Yaskawa INFORM job: pointsclTRJ3.JBI

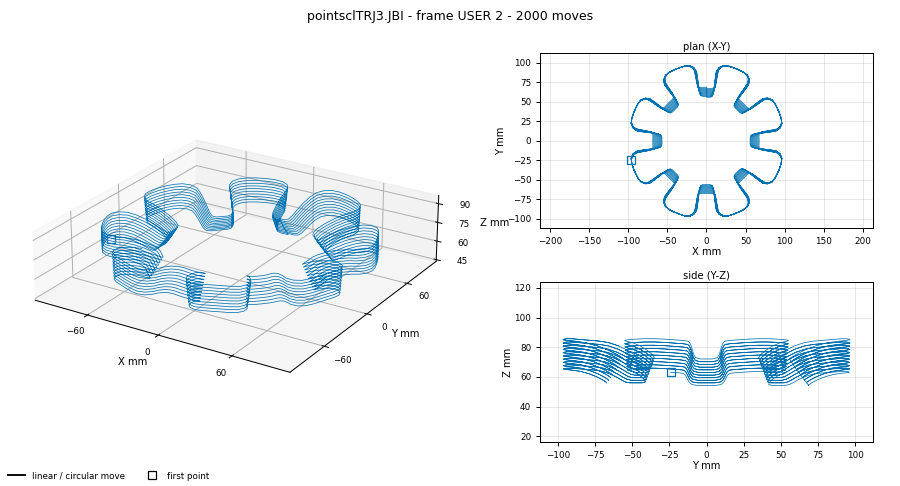
[picture p0: tool path of pointsclTRJ3.JBI in frame USER 2, 2000 of 2000 moves have a stored position in this frame; points joined in program order, loops and branches not executed]
/JOB
//NAME pointsclTRJ3
//POS
///NPOS 2000,0,0,0,0,0
///USER 2
///TOOL 1
///POSTYPE USER
///RECTAN
///RCONF 1,0,0,0,0,0,0,0,0,0,0,0,0,0,0,0,0,0,0,0,0,0,0,0
C00000=-96.154,-24.159,63.210,179.4924,-0.1709,0.0000
C00001=-94.423,-19.246,62.877,-176.7976,1.2873,0.0000
C00002=-90.636,-15.942,62.469,-165.8559,10.6912,0.0000
C00003=-85.405,-14.621,61.698,-164.6923,28.3238,0.0000
C00004=-79.780,-13.569,60.151,-168.6489,33.5433,0.0000
C00005=-74.809,-12.586,58.158,-171.6165,35.6488,0.0000
C00006=-71.127,-11.507,56.252,-173.9501,36.7948,0.0000
C00007=-69.044,-9.699,54.888,-176.7981,37.7947,0.0000
C00008=-68.619,-6.200,54.350,178.5963,38.6094,0.0000
C00009=-68.781,-2.945,54.326,177.6722,38.7088,0.0000
C00010=-68.843,0.000,54.342,179.9995,38.7580,0.0000
C00011=-68.781,2.945,54.326,-177.6718,38.7088,0.0000
C00012=-68.619,6.200,54.350,-178.5977,38.6093,0.0000
C00013=-69.044,9.699,54.888,176.7976,37.7946,0.0000
C00014=-71.127,11.507,56.252,173.9499,36.7948,0.0000
C00015=-74.809,12.586,58.158,171.6165,35.6489,0.0000
C00016=-79.780,13.569,60.151,168.6492,33.5435,0.0000
C00017=-85.405,14.621,61.698,164.6926,28.3243,0.0000
C00018=-90.636,15.942,62.469,165.8558,10.6913,0.0000
C00019=-94.423,19.246,62.877,176.7976,1.2873,0.0000
C00020=-96.154,24.159,63.210,-179.4924,-0.1709,0.0000
C00021=-95.429,29.718,63.547,-178.6193,-0.4469,0.0000
C00022=-93.512,35.416,63.770,-178.6260,-0.4442,0.0000
C00023=-91.166,41.080,63.770,178.7143,0.6573,0.0000
C00024=-88.493,46.465,63.547,178.7076,0.6602,0.0000
C00025=-85.074,50.908,63.210,179.5202,0.2381,0.0000
C00026=-80.376,53.158,62.877,-176.8246,-1.3526,0.0000
C00027=-75.362,52.817,62.469,-162.4707,-2.2128,0.0000
C00028=-70.729,50.052,61.698,-149.5155,9.8553,0.0000
C00029=-66.007,46.818,60.151,-148.1972,15.9457,0.0000
C00030=-61.798,43.998,58.158,-148.3322,19.1679,0.0000
C00031=-58.431,42.158,56.252,-148.7511,21.3364,0.0000
C00032=-55.679,41.963,54.888,-149.5105,23.7114,0.0000
C00033=-52.905,44.137,54.350,-151.2990,27.0505,0.0000
C00034=-50.718,46.553,54.326,-151.7019,27.6849,0.0000
C00035=-48.679,48.679,54.342,-150.4177,26.2748,0.0000
C00036=-46.553,50.718,54.326,-149.2095,24.8209,0.0000
C00037=-44.137,52.905,54.350,-149.7945,25.3228,0.0000
C00038=-41.963,55.680,54.888,-152.9932,27.6813,0.0000
C00039=-42.158,58.431,56.252,-155.4443,28.8948,0.0000
C00040=-43.998,61.798,58.158,-157.7838,29.7283,0.0000
C00041=-46.818,66.007,60.151,-161.4173,30.4455,0.0000
C00042=-50.052,70.729,61.698,-168.6017,29.9881,0.0000
C00043=-52.817,75.362,62.469,177.6796,17.5160,0.0000
C00044=-53.158,80.376,62.877,178.6453,3.1745,0.0000
C00045=-50.908,85.074,63.210,-179.7619,-0.4798,0.0000
C00046=-46.465,88.493,63.547,-179.3396,-1.2923,0.0000
C00047=-41.080,91.166,63.770,-179.3425,-1.2856,0.0000
C00048=-35.416,93.512,63.770,179.5557,1.3739,0.0000
C00049=-29.718,95.429,63.547,179.5530,1.3807,0.0000
C00050=-24.159,96.154,63.210,179.8291,0.5076,0.0000
C00051=-19.246,94.423,62.877,-178.7107,-3.2015,0.0000
C00052=-15.942,90.636,62.469,-168.9825,-13.8937,0.0000
C00053=-14.621,85.405,61.698,-150.8028,-13.4378,0.0000
C00054=-13.569,79.780,60.151,-145.9333,-9.4414,0.0000
C00055=-12.586,74.809,58.158,-144.0591,-6.8041,0.0000
C00056=-11.507,71.127,56.252,-143.0516,-4.8416,0.0000
C00057=-9.699,69.044,54.888,-142.1620,-2.5301,0.0000
C00058=-6.200,68.619,54.350,-141.3823,1.0957,0.0000
C00059=-2.945,68.781,54.326,-141.2681,1.8166,0.0000
C00060=0.000,68.843,54.342,-141.2420,-0.0004,0.0000
C00061=0.000,67.469,56.061,-141.4823,-0.0004,0.0000
C00062=2.820,67.413,56.044,-141.5076,-1.7803,0.0000
C00063=5.989,67.263,56.069,-141.6204,-1.0470,0.0000
C00064=9.441,67.734,56.637,-142.4011,2.5965,0.0000
C00065=11.191,69.937,58.076,-143.2756,4.8842,0.0000
C00066=12.227,73.809,60.085,-144.2799,6.8707,0.0000
C00067=13.183,79.025,62.181,-146.2548,9.6475,0.0000
C00068=14.211,84.918,63.804,-151.9178,13.9840,0.0000
C00069=15.500,90.396,64.610,-174.0678,10.2549,0.0000
C00070=18.832,94.373,65.037,-179.6142,1.0976,0.0000
C00071=23.832,96.213,65.385,179.4380,-1.8355,0.0000
C00072=29.513,95.497,65.736,179.2660,-2.4590,0.0000
C00073=35.347,93.539,65.969,179.2991,-2.3370,0.0000
C00074=41.148,91.136,65.969,-178.8422,2.1478,0.0000
C00075=46.658,88.395,65.736,-178.7792,2.2574,0.0000
C00076=51.181,84.885,65.385,-179.0990,1.6951,0.0000
C00077=53.416,80.048,65.037,179.4966,-1.0488,0.0000
C00078=52.959,74.880,64.610,176.8438,-11.4082,0.0000
C00079=49.997,70.095,63.804,-169.9244,-29.5953,0.0000
C00080=46.557,65.200,62.181,-161.8493,-30.3808,0.0000
C00081=43.545,60.837,60.085,-158.0240,-29.6337,0.0000
C00082=41.540,57.367,58.076,-155.6702,-28.7832,0.0000
C00083=41.220,54.571,56.637,-153.2495,-27.5820,0.0000
C00084=43.327,51.796,56.069,-150.0357,-25.2157,0.0000
C00085=45.674,49.662,56.044,-149.4431,-24.7040,0.0000
C00086=47.708,47.708,56.061,-150.6283,-26.1262,0.0000
C00087=49.662,45.674,56.044,-151.8880,-27.5079,0.0000
C00088=51.797,43.327,56.069,-151.4729,-26.8626,0.0000
C00089=54.571,41.220,56.637,-149.6723,-23.5122,0.0000
C00090=57.367,41.540,58.076,-148.9134,-21.1668,0.0000
C00091=60.837,43.545,60.085,-148.4738,-18.9821,0.0000
C00092=65.200,46.557,62.181,-148.3277,-15.5897,0.0000
C00093=70.095,49.997,63.804,-150.0206,-8.7507,0.0000
C00094=74.880,52.959,64.610,-168.5749,3.0938,0.0000
C00095=80.048,53.416,65.037,-178.9511,0.5034,0.0000
C00096=84.885,51.181,65.385,178.3047,-0.9006,0.0000
C00097=88.395,46.658,65.736,177.7421,-1.2198,0.0000
C00098=91.136,41.148,65.969,177.8518,-1.1570,0.0000
C00099=93.539,35.347,65.969,-177.6628,0.7003,0.0000
C00100=95.497,29.513,65.736,-177.5408,0.7334,0.0000
C00101=96.213,23.832,65.385,-178.1644,0.5617,0.0000
C00102=94.373,18.832,65.037,178.9024,-0.3857,0.0000
C00103=90.396,15.500,64.610,169.6911,-5.8371,0.0000
C00104=84.918,14.211,63.804,164.2377,-27.1799,0.0000
C00105=79.025,13.183,62.181,168.4460,-33.2056,0.0000
C00106=73.809,12.227,60.085,171.5581,-35.4248,0.0000
C00107=69.937,11.191,58.076,173.9145,-36.5694,0.0000
C00108=67.734,9.441,56.637,176.7241,-37.5536,0.0000
C00109=67.263,5.989,56.069,-178.6645,-38.3720,0.0000
C00110=67.413,2.820,56.044,-177.7259,-38.4704,0.0000
C00111=67.469,0.000,56.061,-179.9994,-38.5177,0.0000
C00112=67.413,-2.820,56.044,177.7254,-38.4704,0.0000
C00113=67.263,-5.989,56.069,178.6660,-38.3719,0.0000
C00114=67.734,-9.441,56.637,-176.7236,-37.5535,0.0000
C00115=69.937,-11.191,58.076,-173.9143,-36.5693,0.0000
C00116=73.809,-12.227,60.085,-171.5581,-35.4248,0.0000
C00117=79.025,-13.183,62.181,-168.4462,-33.2058,0.0000
C00118=84.918,-14.211,63.804,-164.2380,-27.1806,0.0000
C00119=90.396,-15.500,64.610,-169.6911,-5.8371,0.0000
C00120=94.373,-18.832,65.037,-178.9024,-0.3857,0.0000
C00121=96.213,-23.832,65.385,178.1644,0.5617,0.0000
C00122=95.497,-29.513,65.736,177.5408,0.7334,0.0000
C00123=93.539,-35.347,65.969,177.6628,0.7003,0.0000
C00124=91.136,-41.148,65.969,-177.8518,-1.1570,0.0000
C00125=88.395,-46.658,65.736,-177.7421,-1.2198,0.0000
C00126=84.885,-51.181,65.385,-178.3047,-0.9006,0.0000
C00127=80.048,-53.416,65.037,178.9511,0.5034,0.0000
C00128=74.880,-52.959,64.610,168.5749,3.0938,0.0000
C00129=70.095,-49.997,63.804,150.0208,-8.7500,0.0000
C00130=65.200,-46.557,62.181,148.3277,-15.5894,0.0000
C00131=60.837,-43.545,60.085,148.4738,-18.9821,0.0000
C00132=57.367,-41.540,58.076,148.9135,-21.1669,0.0000
C00133=54.571,-41.220,56.637,149.6725,-23.5126,0.0000
C00134=51.796,-43.327,56.069,151.4737,-26.8636,0.0000
C00135=49.662,-45.674,56.044,151.8878,-27.5076,0.0000
C00136=47.708,-47.708,56.061,150.6289,-26.1269,0.0000
C00137=45.674,-49.662,56.044,149.4428,-24.7037,0.0000
C00138=43.327,-51.797,56.069,150.0365,-25.2165,0.0000
C00139=41.220,-54.571,56.637,153.2499,-27.5823,0.0000
C00140=41.540,-57.367,58.076,155.6703,-28.7832,0.0000
C00141=43.545,-60.837,60.085,158.0240,-29.6337,0.0000
C00142=46.557,-65.200,62.181,161.8489,-30.3807,0.0000
C00143=49.997,-70.095,63.804,169.9236,-29.5954,0.0000
C00144=52.959,-74.880,64.610,-176.8438,-11.4082,0.0000
C00145=53.416,-80.048,65.037,-179.4966,-1.0488,0.0000
C00146=51.181,-84.885,65.385,179.0990,1.6951,0.0000
C00147=46.658,-88.395,65.736,178.7792,2.2574,0.0000
C00148=41.148,-91.136,65.969,178.8422,2.1478,0.0000
C00149=35.347,-93.539,65.969,-179.2991,-2.3370,0.0000
C00150=29.513,-95.497,65.736,-179.2660,-2.4590,0.0000
C00151=23.832,-96.213,65.385,-179.4380,-1.8355,0.0000
C00152=18.832,-94.373,65.037,179.6142,1.0976,0.0000
C00153=15.500,-90.396,64.610,174.0678,10.2549,0.0000
C00154=14.211,-84.918,63.804,151.9178,13.9840,0.0000
C00155=13.183,-79.025,62.181,146.2548,9.6475,0.0000
C00156=12.227,-73.809,60.085,144.2799,6.8707,0.0000
C00157=11.191,-69.937,58.076,143.2756,4.8842,0.0000
C00158=9.441,-67.734,56.637,142.4011,2.5965,0.0000
C00159=5.989,-67.263,56.069,141.6204,-1.0470,0.0000
C00160=2.820,-67.413,56.044,141.5076,-1.7803,0.0000
C00161=0.000,-67.469,56.061,141.4823,-0.0004,0.0000
C00162=0.000,-67.469,56.061,141.4823,-0.0004,0.0000
C00163=-2.820,-67.413,56.044,141.5076,1.7807,0.0000
C00164=-5.989,-67.263,56.069,141.6205,1.0458,0.0000
C00165=-9.441,-67.734,56.637,142.4012,-2.5969,0.0000
C00166=-11.191,-69.937,58.076,143.2756,-4.8844,0.0000
C00167=-12.227,-73.809,60.085,144.2799,-6.8707,0.0000
C00168=-13.183,-79.025,62.181,146.2546,-9.6473,0.0000
C00169=-14.211,-84.918,63.804,151.9172,-13.9836,0.0000
C00170=-15.500,-90.396,64.610,174.0678,-10.2549,0.0000
C00171=-18.832,-94.373,65.037,179.6142,-1.0976,0.0000
C00172=-23.832,-96.213,65.385,-179.4380,1.8355,0.0000
C00173=-29.513,-95.497,65.736,-179.2660,2.4590,0.0000
C00174=-35.347,-93.539,65.969,-179.2991,2.3370,0.0000
C00175=-41.148,-91.136,65.969,178.8422,-2.1478,0.0000
C00176=-46.658,-88.395,65.736,178.7792,-2.2574,0.0000
C00177=-51.181,-84.885,65.385,179.0990,-1.6951,0.0000
C00178=-53.416,-80.048,65.037,-179.4966,1.0488,0.0000
C00179=-52.959,-74.880,64.610,-176.8438,11.4082,0.0000
C00180=-49.997,-70.095,63.804,169.9244,29.5953,0.0000
C00181=-46.557,-65.200,62.181,161.8493,30.3808,0.0000
C00182=-43.545,-60.837,60.085,158.0240,29.6337,0.0000
C00183=-41.540,-57.367,58.076,155.6702,28.7832,0.0000
C00184=-41.220,-54.571,56.637,153.2495,27.5820,0.0000
C00185=-43.327,-51.796,56.069,150.0357,25.2157,0.0000
C00186=-45.674,-49.662,56.044,149.4431,24.7040,0.0000
C00187=-47.708,-47.708,56.061,150.6283,26.1262,0.0000
C00188=-49.662,-45.674,56.044,151.8880,27.5079,0.0000
C00189=-51.797,-43.327,56.069,151.4729,26.8626,0.0000
C00190=-54.571,-41.220,56.637,149.6723,23.5122,0.0000
C00191=-57.367,-41.540,58.076,148.9134,21.1668,0.0000
C00192=-60.837,-43.545,60.085,148.4738,18.9821,0.0000
C00193=-65.200,-46.557,62.181,148.3277,15.5897,0.0000
C00194=-70.095,-49.997,63.804,150.0206,8.7507,0.0000
C00195=-74.880,-52.959,64.610,168.5749,-3.0938,0.0000
C00196=-80.048,-53.416,65.037,178.9511,-0.5034,0.0000
C00197=-84.885,-51.181,65.385,-178.3047,0.9006,0.0000
C00198=-88.395,-46.658,65.736,-177.7421,1.2198,0.0000
C00199=-91.136,-41.148,65.969,-177.8518,1.1570,0.0000
C00200=-93.539,-35.347,65.969,177.6628,-0.7003,0.0000
C00201=-95.497,-29.513,65.736,177.5408,-0.7334,0.0000
C00202=-96.213,-23.832,65.385,178.1644,-0.5617,0.0000
C00203=-94.373,-18.832,65.037,-178.9024,0.3857,0.0000
C00204=-90.396,-15.500,64.610,-169.6911,5.8371,0.0000
C00205=-84.918,-14.211,63.804,-164.2377,27.1799,0.0000
C00206=-79.025,-13.183,62.181,-168.4460,33.2056,0.0000
C00207=-73.809,-12.227,60.085,-171.5581,35.4248,0.0000
C00208=-69.937,-11.191,58.076,-173.9145,36.5694,0.0000
C00209=-67.734,-9.441,56.637,-176.7241,37.5536,0.0000
C00210=-67.263,-5.989,56.069,178.6645,38.3720,0.0000
C00211=-67.413,-2.820,56.044,177.7259,38.4704,0.0000
C00212=-67.469,0.000,56.061,179.9994,38.5177,0.0000
C00213=-67.413,2.820,56.044,-177.7254,38.4704,0.0000
C00214=-67.263,5.989,56.069,-178.6660,38.3719,0.0000
C00215=-67.734,9.441,56.637,176.7236,37.5535,0.0000
C00216=-69.937,11.191,58.076,173.9143,36.5693,0.0000
C00217=-73.809,12.227,60.085,171.5581,35.4248,0.0000
C00218=-79.025,13.183,62.181,168.4462,33.2058,0.0000
C00219=-84.918,14.211,63.804,164.2380,27.1806,0.0000
C00220=-90.396,15.500,64.610,169.6911,5.8371,0.0000
C00221=-94.373,18.832,65.037,178.9024,0.3857,0.0000
C00222=-96.213,23.832,65.385,-178.1644,-0.5617,0.0000
C00223=-95.497,29.513,65.736,-177.5408,-0.7334,0.0000
C00224=-93.539,35.347,65.969,-177.6628,-0.7003,0.0000
C00225=-91.136,41.148,65.969,177.8518,1.1570,0.0000
C00226=-88.395,46.658,65.736,177.7421,1.2198,0.0000
C00227=-84.885,51.181,65.385,178.3047,0.9006,0.0000
C00228=-80.048,53.416,65.037,-178.9511,-0.5034,0.0000
C00229=-74.880,52.959,64.610,-168.5749,-3.0938,0.0000
C00230=-70.095,49.997,63.804,-150.0208,8.7500,0.0000
C00231=-65.200,46.557,62.181,-148.3277,15.5894,0.0000
C00232=-60.837,43.545,60.085,-148.4738,18.9821,0.0000
C00233=-57.367,41.540,58.076,-148.9135,21.1669,0.0000
C00234=-54.571,41.220,56.637,-149.6725,23.5126,0.0000
C00235=-51.796,43.327,56.069,-151.4737,26.8636,0.0000
C00236=-49.662,45.674,56.044,-151.8878,27.5076,0.0000
C00237=-47.708,47.708,56.061,-150.6289,26.1269,0.0000
C00238=-45.674,49.662,56.044,-149.4428,24.7037,0.0000
C00239=-43.327,51.797,56.069,-150.0365,25.2165,0.0000
C00240=-41.220,54.571,56.637,-153.2499,27.5823,0.0000
C00241=-41.540,57.367,58.076,-155.6703,28.7832,0.0000
C00242=-43.545,60.837,60.085,-158.0240,29.6337,0.0000
C00243=-46.557,65.200,62.181,-161.8489,30.3807,0.0000
C00244=-49.997,70.095,63.804,-169.9236,29.5954,0.0000
C00245=-52.959,74.880,64.610,176.8438,11.4082,0.0000
C00246=-53.416,80.048,65.037,179.4966,1.0488,0.0000
C00247=-51.181,84.885,65.385,-179.0990,-1.6951,0.0000
C00248=-46.658,88.395,65.736,-178.7792,-2.2574,0.0000
C00249=-41.148,91.136,65.969,-178.8422,-2.1478,0.0000
C00250=-35.347,93.539,65.969,179.2991,2.3370,0.0000
C00251=-29.513,95.497,65.736,179.2660,2.4590,0.0000
C00252=-23.832,96.213,65.385,179.4380,1.8355,0.0000
C00253=-18.832,94.373,65.037,-179.6142,-1.0976,0.0000
C00254=-15.500,90.396,64.610,-174.0678,-10.2549,0.0000
C00255=-14.211,84.918,63.804,-151.9172,-13.9836,0.0000
C00256=-13.183,79.025,62.181,-146.2546,-9.6473,0.0000
C00257=-12.227,73.809,60.085,-144.2799,-6.8707,0.0000
C00258=-11.191,69.937,58.076,-143.2756,-4.8844,0.0000
C00259=-9.441,67.734,56.637,-142.4012,-2.5969,0.0000
C00260=-5.989,67.263,56.069,-141.6205,1.0458,0.0000
C00261=-2.820,67.413,56.044,-141.5076,1.7807,0.0000
C00262=0.000,67.469,56.061,-141.4823,-0.0004,0.0000
C00263=0.000,66.107,57.788,-141.7677,-0.0005,0.0000
C00264=2.695,66.055,57.771,-141.7921,-1.7411,0.0000
C00265=5.779,65.917,57.797,-141.9032,-1.0017,0.0000
C00266=9.185,66.436,58.394,-142.6835,2.6509,0.0000
C00267=10.880,68.762,59.909,-143.5425,4.9131,0.0000
C00268=11.874,72.826,62.021,-144.5463,6.9278,0.0000
C00269=12.805,78.288,64.219,-146.6451,9.8629,0.0000
C00270=13.814,84.445,65.915,-153.3894,14.5606,0.0000
C00271=15.073,90.163,66.756,-176.7990,6.8806,0.0000
C00272=18.432,94.325,67.200,179.8056,-0.6227,0.0000
C00273=23.517,96.271,67.561,179.1749,-2.9305,0.0000
C00274=29.315,95.562,67.927,179.0643,-3.3741,0.0000
C00275=35.280,93.564,68.167,179.1110,-3.1790,0.0000
C00276=41.213,91.107,68.167,-178.3786,2.8755,0.0000
C00277=46.844,88.301,67.927,-178.2733,3.0464,0.0000
C00278=51.445,84.703,67.561,-178.5096,2.6549,0.0000
C00279=53.664,79.731,67.200,-179.6972,0.5778,0.0000
C00280=53.097,74.413,66.756,177.3712,-7.1180,0.0000
C00281=49.944,69.479,65.915,-171.5349,-28.9684,0.0000
C00282=46.303,64.413,64.219,-162.3452,-30.2755,0.0000
C00283=43.100,59.892,62.021,-158.2955,-29.5017,0.0000
C00284=40.929,56.315,59.909,-155.9227,-28.6330,0.0000
C00285=40.483,53.472,58.394,-153.5346,-27.4456,0.0000
C00286=42.524,50.697,57.797,-150.3130,-25.0779,0.0000
C00287=44.802,48.614,57.771,-149.7172,-24.5616,0.0000
C00288=46.745,46.745,57.788,-150.8781,-25.9501,0.0000
C00289=48.613,44.802,57.771,-152.1106,-27.2998,0.0000
C00290=50.697,42.524,57.797,-151.6894,-26.6512,0.0000
C00291=53.472,40.483,58.395,-149.8793,-23.2967,0.0000
C00292=56.315,40.929,59.909,-149.1208,-20.9821,0.0000
C00293=59.892,43.100,62.021,-148.6591,-18.7760,0.0000
C00294=64.413,46.303,64.219,-148.5069,-15.1841,0.0000
C00295=69.479,49.944,65.915,-150.7646,-7.4003,0.0000
C00296=74.413,53.097,66.756,-172.8746,2.6086,0.0000
C00297=79.731,53.664,67.200,179.4222,-0.3028,0.0000
C00298=84.703,51.445,67.561,177.3442,-1.4888,0.0000
C00299=88.301,46.844,67.927,176.9523,-1.7243,0.0000
C00300=91.107,41.213,68.167,177.1233,-1.6193,0.0000
C00301=93.564,35.280,68.167,-176.8206,0.8876,0.0000
C00302=95.562,29.315,67.927,-176.6255,0.9341,0.0000
C00303=96.271,23.517,67.561,-177.0692,0.8240,0.0000
C00304=94.325,18.432,67.200,-179.3773,0.1944,0.0000
C00305=90.163,15.073,66.756,173.1087,-3.1780,0.0000
C00306=84.445,13.814,65.915,163.8003,-25.6923,0.0000
C00307=78.288,12.805,64.219,168.2420,-32.7993,0.0000
C00308=72.826,11.874,62.021,171.5162,-35.1564,0.0000
C00309=68.762,10.880,59.909,173.8995,-36.3021,0.0000
C00310=66.436,9.185,58.394,176.6682,-37.2698,0.0000
C00311=65.917,5.779,57.797,-178.7272,-38.0899,0.0000
C00312=66.055,2.695,57.771,-177.7847,-38.1871,0.0000
C00313=66.107,0.000,57.788,-179.9993,-38.2323,0.0000
C00314=66.055,-2.695,57.771,177.7841,-38.1871,0.0000
C00315=65.917,-5.780,57.797,178.7287,-38.0898,0.0000
C00316=66.436,-9.185,58.395,-176.6677,-37.2697,0.0000
C00317=68.762,-10.880,59.909,-173.8994,-36.3021,0.0000
C00318=72.826,-11.874,62.021,-171.5162,-35.1564,0.0000
C00319=78.288,-12.805,64.219,-168.2422,-32.7995,0.0000
C00320=84.445,-13.814,65.915,-163.8006,-25.6930,0.0000
C00321=90.163,-15.073,66.756,-173.1087,-3.1780,0.0000
C00322=94.325,-18.432,67.200,179.3773,0.1944,0.0000
C00323=96.271,-23.517,67.561,177.0692,0.8240,0.0000
C00324=95.562,-29.315,67.927,176.6255,0.9341,0.0000
C00325=93.564,-35.280,68.167,176.8206,0.8876,0.0000
C00326=91.107,-41.213,68.167,-177.1233,-1.6193,0.0000
C00327=88.301,-46.844,67.927,-176.9523,-1.7243,0.0000
C00328=84.703,-51.445,67.561,-177.3442,-1.4888,0.0000
C00329=79.731,-53.664,67.200,-179.4222,-0.3028,0.0000
C00330=74.413,-53.097,66.756,172.8746,2.6086,0.0000
C00331=69.479,-49.944,65.915,150.7649,-7.3996,0.0000
C00332=64.413,-46.303,64.219,148.5069,-15.1838,0.0000
C00333=59.892,-43.100,62.021,148.6592,-18.7760,0.0000
C00334=56.315,-40.929,59.909,149.1208,-20.9822,0.0000
C00335=53.472,-40.483,58.394,149.8795,-23.2971,0.0000
C00336=50.697,-42.524,57.797,151.6901,-26.6522,0.0000
C00337=48.614,-44.802,57.771,152.1103,-27.2994,0.0000
C00338=46.745,-46.745,57.788,150.8789,-25.9509,0.0000
C00339=44.802,-48.613,57.771,149.7168,-24.5613,0.0000
C00340=42.524,-50.697,57.797,150.3139,-25.0788,0.0000
C00341=40.483,-53.472,58.395,153.5350,-27.4458,0.0000
C00342=40.929,-56.315,59.909,155.9228,-28.6331,0.0000
C00343=43.100,-59.892,62.021,158.2955,-29.5017,0.0000
C00344=46.303,-64.413,64.219,162.3449,-30.2755,0.0000
C00345=49.944,-69.479,65.915,171.5341,-28.9686,0.0000
C00346=53.097,-74.413,66.756,-177.3712,-7.1180,0.0000
C00347=53.664,-79.731,67.200,179.6972,0.5778,0.0000
C00348=51.445,-84.703,67.561,178.5096,2.6549,0.0000
C00349=46.844,-88.301,67.927,178.2733,3.0464,0.0000
C00350=41.213,-91.107,68.167,178.3786,2.8755,0.0000
C00351=35.280,-93.564,68.167,-179.1110,-3.1790,0.0000
C00352=29.315,-95.562,67.927,-179.0643,-3.3741,0.0000
C00353=23.517,-96.271,67.561,-179.1749,-2.9305,0.0000
C00354=18.432,-94.325,67.200,-179.8056,-0.6227,0.0000
C00355=15.073,-90.163,66.756,176.7990,6.8806,0.0000
C00356=13.814,-84.445,65.915,153.3894,14.5606,0.0000
C00357=12.805,-78.288,64.219,146.6451,9.8629,0.0000
C00358=11.874,-72.826,62.021,144.5463,6.9278,0.0000
C00359=10.880,-68.762,59.909,143.5425,4.9131,0.0000
C00360=9.185,-66.436,58.394,142.6835,2.6509,0.0000
C00361=5.779,-65.917,57.797,141.9032,-1.0017,0.0000
C00362=2.695,-66.055,57.771,141.7921,-1.7411,0.0000
C00363=0.000,-66.107,57.788,141.7677,-0.0005,0.0000
C00364=0.000,-66.107,57.788,141.7677,-0.0005,0.0000
C00365=-2.695,-66.055,57.771,141.7920,1.7416,0.0000
C00366=-5.780,-65.917,57.797,141.9033,1.0005,0.0000
C00367=-9.185,-66.436,58.395,142.6836,-2.6513,0.0000
C00368=-10.880,-68.762,59.909,143.5425,-4.9132,0.0000
C00369=-11.874,-72.826,62.021,144.5463,-6.9278,0.0000
C00370=-12.805,-78.288,64.219,146.6449,-9.8627,0.0000
C00371=-13.814,-84.445,65.915,153.3887,-14.5602,0.0000
C00372=-15.073,-90.163,66.756,176.7990,-6.8806,0.0000
C00373=-18.432,-94.325,67.200,-179.8056,0.6227,0.0000
C00374=-23.517,-96.271,67.561,-179.1749,2.9305,0.0000
C00375=-29.315,-95.562,67.927,-179.0643,3.3741,0.0000
C00376=-35.280,-93.564,68.167,-179.1110,3.1790,0.0000
C00377=-41.213,-91.107,68.167,178.3786,-2.8755,0.0000
C00378=-46.844,-88.301,67.927,178.2733,-3.0464,0.0000
C00379=-51.445,-84.703,67.561,178.5096,-2.6549,0.0000
C00380=-53.664,-79.731,67.200,179.6972,-0.5778,0.0000
C00381=-53.097,-74.413,66.756,-177.3712,7.1180,0.0000
C00382=-49.944,-69.479,65.915,171.5349,28.9684,0.0000
C00383=-46.303,-64.413,64.219,162.3452,30.2755,0.0000
C00384=-43.100,-59.892,62.021,158.2955,29.5017,0.0000
C00385=-40.929,-56.315,59.909,155.9227,28.6330,0.0000
C00386=-40.483,-53.472,58.394,153.5346,27.4456,0.0000
C00387=-42.524,-50.697,57.797,150.3130,25.0779,0.0000
C00388=-44.802,-48.614,57.771,149.7172,24.5616,0.0000
C00389=-46.745,-46.745,57.788,150.8781,25.9501,0.0000
C00390=-48.613,-44.802,57.771,152.1106,27.2998,0.0000
C00391=-50.697,-42.524,57.797,151.6894,26.6512,0.0000
C00392=-53.472,-40.483,58.395,149.8793,23.2967,0.0000
C00393=-56.315,-40.929,59.909,149.1208,20.9821,0.0000
C00394=-59.892,-43.100,62.021,148.6591,18.7760,0.0000
C00395=-64.413,-46.303,64.219,148.5069,15.1841,0.0000
C00396=-69.479,-49.944,65.915,150.7646,7.4003,0.0000
C00397=-74.413,-53.097,66.756,172.8746,-2.6086,0.0000
C00398=-79.731,-53.664,67.200,-179.4222,0.3028,0.0000
C00399=-84.703,-51.445,67.561,-177.3442,1.4888,0.0000
C00400=-88.301,-46.844,67.927,-176.9523,1.7243,0.0000
C00401=-91.107,-41.213,68.167,-177.1233,1.6193,0.0000
C00402=-93.564,-35.280,68.167,176.8206,-0.8876,0.0000
C00403=-95.562,-29.315,67.927,176.6255,-0.9341,0.0000
C00404=-96.271,-23.517,67.561,177.0692,-0.8240,0.0000
C00405=-94.325,-18.432,67.200,179.3773,-0.1944,0.0000
C00406=-90.163,-15.073,66.756,-173.1087,3.1780,0.0000
C00407=-84.445,-13.814,65.915,-163.8003,25.6923,0.0000
C00408=-78.288,-12.805,64.219,-168.2420,32.7993,0.0000
C00409=-72.826,-11.874,62.021,-171.5162,35.1564,0.0000
C00410=-68.762,-10.880,59.909,-173.8995,36.3021,0.0000
C00411=-66.436,-9.185,58.394,-176.6682,37.2698,0.0000
C00412=-65.917,-5.779,57.797,178.7272,38.0899,0.0000
C00413=-66.055,-2.695,57.771,177.7847,38.1871,0.0000
C00414=-66.107,0.000,57.788,179.9993,38.2323,0.0000
C00415=-66.055,2.695,57.771,-177.7841,38.1871,0.0000
C00416=-65.917,5.780,57.797,-178.7287,38.0898,0.0000
C00417=-66.436,9.185,58.395,176.6677,37.2697,0.0000
C00418=-68.762,10.880,59.909,173.8994,36.3021,0.0000
C00419=-72.826,11.874,62.021,171.5162,35.1564,0.0000
C00420=-78.288,12.805,64.219,168.2422,32.7995,0.0000
C00421=-84.445,13.814,65.915,163.8006,25.6930,0.0000
C00422=-90.163,15.073,66.756,173.1087,3.1780,0.0000
C00423=-94.325,18.432,67.200,-179.3773,-0.1944,0.0000
C00424=-96.271,23.517,67.561,-177.0692,-0.8240,0.0000
C00425=-95.562,29.315,67.927,-176.6255,-0.9341,0.0000
C00426=-93.564,35.280,68.167,-176.8206,-0.8876,0.0000
C00427=-91.107,41.213,68.167,177.1233,1.6193,0.0000
C00428=-88.301,46.844,67.927,176.9523,1.7243,0.0000
C00429=-84.703,51.445,67.561,177.3442,1.4888,0.0000
C00430=-79.731,53.664,67.200,179.4222,0.3028,0.0000
C00431=-74.413,53.097,66.756,-172.8746,-2.6086,0.0000
C00432=-69.479,49.944,65.915,-150.7649,7.3996,0.0000
C00433=-64.413,46.303,64.219,-148.5069,15.1838,0.0000
C00434=-59.892,43.100,62.021,-148.6592,18.7760,0.0000
C00435=-56.315,40.929,59.909,-149.1208,20.9822,0.0000
C00436=-53.472,40.483,58.394,-149.8795,23.2971,0.0000
C00437=-50.697,42.524,57.797,-151.6901,26.6522,0.0000
C00438=-48.614,44.802,57.771,-152.1103,27.2994,0.0000
C00439=-46.745,46.745,57.788,-150.8789,25.9509,0.0000
C00440=-44.802,48.613,57.771,-149.7168,24.5613,0.0000
C00441=-42.524,50.697,57.797,-150.3139,25.0788,0.0000
C00442=-40.483,53.472,58.395,-153.5350,27.4458,0.0000
C00443=-40.929,56.315,59.909,-155.9228,28.6331,0.0000
C00444=-43.100,59.892,62.021,-158.2955,29.5017,0.0000
C00445=-46.303,64.413,64.219,-162.3449,30.2755,0.0000
C00446=-49.944,69.479,65.915,-171.5341,28.9686,0.0000
C00447=-53.097,74.413,66.756,177.3712,7.1180,0.0000
C00448=-53.664,79.731,67.200,-179.6972,-0.5778,0.0000
C00449=-51.445,84.703,67.561,-178.5096,-2.6549,0.0000
C00450=-46.844,88.301,67.927,-178.2733,-3.0464,0.0000
C00451=-41.213,91.107,68.167,-178.3786,-2.8755,0.0000
C00452=-35.280,93.564,68.167,179.1110,3.1790,0.0000
C00453=-29.315,95.562,67.927,179.0643,3.3741,0.0000
C00454=-23.517,96.271,67.561,179.1749,2.9305,0.0000
C00455=-18.432,94.325,67.200,179.8056,0.6227,0.0000
C00456=-15.073,90.163,66.756,-176.7990,-6.8806,0.0000
C00457=-13.814,84.445,65.915,-153.3887,-14.5602,0.0000
C00458=-12.805,78.288,64.219,-146.6449,-9.8627,0.0000
C00459=-11.874,72.826,62.021,-144.5463,-6.9278,0.0000
C00460=-10.880,68.762,59.909,-143.5425,-4.9132,0.0000
C00461=-9.185,66.436,58.395,-142.6836,-2.6513,0.0000
C00462=-5.780,65.917,57.797,-141.9033,1.0005,0.0000
C00463=-2.695,66.055,57.771,-141.7920,1.7416,0.0000
C00464=0.000,66.107,57.788,-141.7677,-0.0005,0.0000
C00465=0.000,64.758,59.526,-142.0985,-0.0006,0.0000
C00466=2.572,64.710,59.508,-142.1219,-1.6987,0.0000
C00467=5.572,64.584,59.535,-142.2312,-0.9609,0.0000
C00468=8.932,65.152,60.163,-143.0096,2.6933,0.0000
C00469=10.572,67.603,61.754,-143.8534,4.9293,0.0000
C00470=11.527,71.864,63.969,-144.8604,6.9774,0.0000
C00471=12.439,77.571,66.266,-147.1134,10.0930,0.0000
C00472=13.430,83.988,68.033,-155.3821,15.1332,0.0000
C00473=14.662,89.940,68.906,-178.5212,3.8469,0.0000
C00474=18.048,94.279,69.366,179.4400,-1.9851,0.0000
C00475=23.215,96.325,69.740,179.0015,-3.8187,0.0000
C00476=29.126,95.625,70.117,178.9266,-4.1371,0.0000
C00477=35.216,93.589,70.366,178.9774,-3.9012,0.0000
C00478=41.276,91.079,70.366,-177.9608,3.4799,0.0000
C00479=47.022,88.212,70.117,-177.8292,3.6823,0.0000
C00480=51.697,84.528,69.740,-178.0023,3.4047,0.0000
C00481=53.903,79.427,69.366,-178.9918,1.7994,0.0000
C00482=53.229,73.964,68.906,178.3212,-3.7641,0.0000
C00483=49.892,68.885,68.033,-173.5159,-27.9656,0.0000
C00484=46.056,63.647,66.266,-162.9163,-30.1272,0.0000
C00485=42.664,58.966,63.969,-158.6013,-29.3323,0.0000
C00486=40.327,55.279,61.754,-156.2029,-28.4444,0.0000
C00487=39.754,52.385,60.163,-153.8484,-27.2716,0.0000
C00488=41.728,49.608,59.535,-150.6259,-24.9083,0.0000
C00489=43.938,47.576,59.508,-150.0322,-24.3934,0.0000
C00490=45.791,45.791,59.526,-151.1670,-25.7453,0.0000
C00491=47.575,43.938,59.508,-152.3699,-27.0604,0.0000
C00492=49.608,41.728,59.535,-151.9475,-26.4149,0.0000
C00493=52.385,39.754,60.163,-150.1310,-23.0634,0.0000
C00494=55.279,40.327,61.754,-149.3729,-20.7804,0.0000
C00495=58.966,42.664,63.969,-148.8882,-18.5467,0.0000
C00496=63.647,46.056,66.266,-148.7380,-14.7196,0.0000
C00497=68.885,49.892,68.033,-151.8815,-5.7249,0.0000
C00498=73.964,53.229,68.906,-176.2343,1.6751,0.0000
C00499=79.427,53.903,69.366,178.2003,-1.0077,0.0000
C00500=84.528,51.697,69.740,176.5933,-1.9942,0.0000
C00501=88.212,47.022,70.117,176.3150,-2.1663,0.0000
C00502=91.079,41.276,70.366,176.5179,-2.0355,0.0000
C00503=93.589,35.216,70.366,-176.0982,1.0202,0.0000
C00504=95.625,29.126,70.117,-175.8622,1.0706,0.0000
C00505=96.325,23.215,69.740,-176.1807,0.9963,0.0000
C00506=94.279,18.048,69.366,-178.0148,0.5597,0.0000
C00507=89.940,14.662,68.906,176.1518,-1.4755,0.0000
C00508=83.988,13.430,68.033,163.4332,-23.7107,0.0000
C00509=77.571,12.439,66.266,168.0321,-32.3152,0.0000
C00510=71.864,11.527,63.969,171.4883,-34.8415,0.0000
C00511=67.603,10.572,61.754,173.9037,-35.9920,0.0000
C00512=65.152,8.932,60.163,176.6294,-36.9427,0.0000
C00513=64.584,5.572,59.535,-178.7845,-37.7626,0.0000
C00514=64.710,2.572,59.508,-177.8483,-37.8585,0.0000
C00515=64.758,0.000,59.526,-179.9992,-37.9015,0.0000
C00516=64.710,-2.572,59.508,177.8476,-37.8585,0.0000
C00517=64.584,-5.572,59.535,178.7860,-37.7625,0.0000
C00518=65.152,-8.932,60.163,-176.6289,-36.9426,0.0000
C00519=67.603,-10.572,61.754,-173.9036,-35.9920,0.0000
C00520=71.864,-11.527,63.969,-171.4883,-34.8415,0.0000
C00521=77.571,-12.439,66.266,-168.0323,-32.3154,0.0000
C00522=83.988,-13.430,68.033,-163.4334,-23.7115,0.0000
C00523=89.940,-14.662,68.906,-176.1518,-1.4755,0.0000
C00524=94.279,-18.048,69.366,178.0148,0.5597,0.0000
C00525=96.325,-23.215,69.740,176.1807,0.9963,0.0000
C00526=95.625,-29.126,70.117,175.8622,1.0706,0.0000
C00527=93.589,-35.216,70.366,176.0982,1.0202,0.0000
C00528=91.079,-41.276,70.366,-176.5179,-2.0355,0.0000
C00529=88.212,-47.022,70.117,-176.3150,-2.1663,0.0000
C00530=84.528,-51.697,69.740,-176.5933,-1.9942,0.0000
C00531=79.427,-53.903,69.366,-178.2003,-1.0077,0.0000
C00532=73.964,-53.229,68.906,176.2343,1.6751,0.0000
C00533=68.885,-49.892,68.033,151.8818,-5.7242,0.0000
C00534=63.647,-46.056,66.266,148.7380,-14.7193,0.0000
C00535=58.966,-42.664,63.969,148.8883,-18.5467,0.0000
C00536=55.279,-40.327,61.754,149.3730,-20.7805,0.0000
C00537=52.385,-39.754,60.163,150.1312,-23.0638,0.0000
C00538=49.608,-41.728,59.535,151.9483,-26.4159,0.0000
C00539=47.576,-43.938,59.508,152.3695,-27.0599,0.0000
C00540=45.791,-45.791,59.526,151.1678,-25.7463,0.0000
C00541=43.938,-47.575,59.508,150.0318,-24.3930,0.0000
C00542=41.728,-49.608,59.535,150.6268,-24.9092,0.0000
C00543=39.754,-52.385,60.163,153.8488,-27.2719,0.0000
C00544=40.327,-55.279,61.754,156.2030,-28.4445,0.0000
C00545=42.664,-58.966,63.969,158.6013,-29.3323,0.0000
C00546=46.056,-63.647,66.266,162.9160,-30.1271,0.0000
C00547=49.892,-68.885,68.033,173.5151,-27.9659,0.0000
C00548=53.229,-73.964,68.906,-178.3212,-3.7641,0.0000
C00549=53.903,-79.427,69.366,178.9918,1.7994,0.0000
C00550=51.697,-84.528,69.740,178.0023,3.4047,0.0000
C00551=47.022,-88.212,70.117,177.8292,3.6823,0.0000
C00552=41.276,-91.079,70.366,177.9608,3.4799,0.0000
C00553=35.216,-93.589,70.366,-178.9774,-3.9012,0.0000
C00554=29.126,-95.625,70.117,-178.9266,-4.1371,0.0000
C00555=23.215,-96.325,69.740,-179.0015,-3.8187,0.0000
C00556=18.048,-94.279,69.366,-179.4400,-1.9851,0.0000
C00557=14.662,-89.940,68.906,178.5212,3.8469,0.0000
C00558=13.430,-83.988,68.033,155.3821,15.1332,0.0000
C00559=12.439,-77.571,66.266,147.1134,10.0930,0.0000
C00560=11.527,-71.864,63.969,144.8604,6.9774,0.0000
C00561=10.572,-67.603,61.754,143.8534,4.9293,0.0000
C00562=8.932,-65.152,60.163,143.0096,2.6933,0.0000
C00563=5.572,-64.584,59.535,142.2312,-0.9609,0.0000
C00564=2.572,-64.710,59.508,142.1219,-1.6987,0.0000
C00565=0.000,-64.758,59.526,142.0985,-0.0006,0.0000
C00566=0.000,-64.758,59.526,142.0985,-0.0006,0.0000
C00567=-2.572,-64.710,59.508,142.1219,1.6993,0.0000
C00568=-5.572,-64.584,59.535,142.2313,0.9597,0.0000
C00569=-8.932,-65.152,60.163,143.0097,-2.6937,0.0000
C00570=-10.572,-67.603,61.754,143.8534,-4.9294,0.0000
C00571=-11.527,-71.864,63.969,144.8604,-6.9774,0.0000
C00572=-12.439,-77.571,66.266,147.1132,-10.0928,0.0000
C00573=-13.430,-83.988,68.033,155.3813,-15.1329,0.0000
C00574=-14.662,-89.940,68.906,178.5212,-3.8469,0.0000
C00575=-18.048,-94.279,69.366,-179.4400,1.9851,0.0000
C00576=-23.215,-96.325,69.740,-179.0015,3.8187,0.0000
C00577=-29.126,-95.625,70.117,-178.9266,4.1371,0.0000
C00578=-35.216,-93.589,70.366,-178.9774,3.9012,0.0000
C00579=-41.276,-91.079,70.366,177.9608,-3.4799,0.0000
C00580=-47.022,-88.212,70.117,177.8292,-3.6823,0.0000
C00581=-51.697,-84.528,69.740,178.0023,-3.4047,0.0000
C00582=-53.903,-79.427,69.366,178.9918,-1.7994,0.0000
C00583=-53.229,-73.964,68.906,-178.3212,3.7641,0.0000
C00584=-49.892,-68.885,68.033,173.5159,27.9656,0.0000
C00585=-46.056,-63.647,66.266,162.9163,30.1272,0.0000
C00586=-42.664,-58.966,63.969,158.6013,29.3323,0.0000
C00587=-40.327,-55.279,61.754,156.2029,28.4444,0.0000
C00588=-39.754,-52.385,60.163,153.8484,27.2716,0.0000
C00589=-41.728,-49.608,59.535,150.6259,24.9083,0.0000
C00590=-43.938,-47.576,59.508,150.0322,24.3934,0.0000
C00591=-45.791,-45.791,59.526,151.1670,25.7453,0.0000
C00592=-47.575,-43.938,59.508,152.3699,27.0604,0.0000
C00593=-49.608,-41.728,59.535,151.9475,26.4149,0.0000
C00594=-52.385,-39.754,60.163,150.1310,23.0634,0.0000
C00595=-55.279,-40.327,61.754,149.3729,20.7804,0.0000
C00596=-58.966,-42.664,63.969,148.8882,18.5467,0.0000
C00597=-63.647,-46.056,66.266,148.7380,14.7196,0.0000
C00598=-68.885,-49.892,68.033,151.8815,5.7249,0.0000
C00599=-73.964,-53.229,68.906,176.2343,-1.6751,0.0000
C00600=-79.427,-53.903,69.366,-178.2003,1.0077,0.0000
C00601=-84.528,-51.697,69.740,-176.5933,1.9942,0.0000
C00602=-88.212,-47.022,70.117,-176.3150,2.1663,0.0000
C00603=-91.079,-41.276,70.366,-176.5179,2.0355,0.0000
C00604=-93.589,-35.216,70.366,176.0982,-1.0202,0.0000
C00605=-95.625,-29.126,70.117,175.8622,-1.0706,0.0000
C00606=-96.325,-23.215,69.740,176.1807,-0.9963,0.0000
C00607=-94.279,-18.048,69.366,178.0148,-0.5597,0.0000
C00608=-89.940,-14.662,68.906,-176.1518,1.4755,0.0000
C00609=-83.988,-13.430,68.033,-163.4332,23.7107,0.0000
C00610=-77.571,-12.439,66.266,-168.0321,32.3152,0.0000
C00611=-71.864,-11.527,63.969,-171.4883,34.8415,0.0000
C00612=-67.603,-10.572,61.754,-173.9037,35.9920,0.0000
C00613=-65.152,-8.932,60.163,-176.6294,36.9427,0.0000
C00614=-64.584,-5.572,59.535,178.7845,37.7626,0.0000
C00615=-64.710,-2.572,59.508,177.8483,37.8585,0.0000
C00616=-64.758,0.000,59.526,179.9992,37.9015,0.0000
C00617=-64.710,2.572,59.508,-177.8476,37.8585,0.0000
C00618=-64.584,5.572,59.535,-178.7860,37.7625,0.0000
C00619=-65.152,8.932,60.163,176.6289,36.9426,0.0000
C00620=-67.603,10.572,61.754,173.9036,35.9920,0.0000
C00621=-71.864,11.527,63.969,171.4883,34.8415,0.0000
C00622=-77.571,12.439,66.266,168.0323,32.3154,0.0000
C00623=-83.988,13.430,68.033,163.4334,23.7115,0.0000
C00624=-89.940,14.662,68.906,176.1518,1.4755,0.0000
C00625=-94.279,18.048,69.366,-178.0148,-0.5597,0.0000
C00626=-96.325,23.215,69.740,-176.1807,-0.9963,0.0000
C00627=-95.625,29.126,70.117,-175.8622,-1.0706,0.0000
C00628=-93.589,35.216,70.366,-176.0982,-1.0202,0.0000
C00629=-91.079,41.276,70.366,176.5179,2.0355,0.0000
C00630=-88.212,47.022,70.117,176.3150,2.1663,0.0000
C00631=-84.528,51.697,69.740,176.5933,1.9942,0.0000
C00632=-79.427,53.903,69.366,178.2003,1.0077,0.0000
C00633=-73.964,53.229,68.906,-176.2343,-1.6751,0.0000
C00634=-68.885,49.892,68.033,-151.8818,5.7242,0.0000
C00635=-63.647,46.056,66.266,-148.7380,14.7193,0.0000
C00636=-58.966,42.664,63.969,-148.8883,18.5467,0.0000
C00637=-55.279,40.327,61.754,-149.3730,20.7805,0.0000
C00638=-52.385,39.754,60.163,-150.1312,23.0638,0.0000
C00639=-49.608,41.728,59.535,-151.9483,26.4159,0.0000
C00640=-47.576,43.938,59.508,-152.3695,27.0599,0.0000
C00641=-45.791,45.791,59.526,-151.1678,25.7463,0.0000
C00642=-43.938,47.575,59.508,-150.0318,24.3930,0.0000
C00643=-41.728,49.608,59.535,-150.6268,24.9092,0.0000
C00644=-39.754,52.385,60.163,-153.8488,27.2719,0.0000
C00645=-40.327,55.279,61.754,-156.2030,28.4445,0.0000
C00646=-42.664,58.966,63.969,-158.6013,29.3323,0.0000
C00647=-46.056,63.647,66.266,-162.9160,30.1271,0.0000
C00648=-49.892,68.885,68.033,-173.5151,27.9659,0.0000
C00649=-53.229,73.964,68.906,178.3212,3.7641,0.0000
C00650=-53.903,79.427,69.366,-178.9918,-1.7994,0.0000
C00651=-51.697,84.528,69.740,-178.0023,-3.4047,0.0000
C00652=-47.022,88.212,70.117,-177.8292,-3.6823,0.0000
C00653=-41.276,91.079,70.366,-177.9608,-3.4799,0.0000
C00654=-35.216,93.589,70.366,178.9774,3.9012,0.0000
C00655=-29.126,95.625,70.117,178.9266,4.1371,0.0000
C00656=-23.215,96.325,69.740,179.0015,3.8187,0.0000
C00657=-18.048,94.279,69.366,179.4400,1.9851,0.0000
C00658=-14.662,89.940,68.906,-178.5212,-3.8469,0.0000
C00659=-13.430,83.988,68.033,-155.3813,-15.1329,0.0000
C00660=-12.439,77.571,66.266,-147.1132,-10.0928,0.0000
C00661=-11.527,71.864,63.969,-144.8604,-6.9774,0.0000
C00662=-10.572,67.603,61.754,-143.8534,-4.9294,0.0000
C00663=-8.932,65.152,60.163,-143.0097,-2.6937,0.0000
C00664=-5.572,64.584,59.535,-142.2313,0.9597,0.0000
C00665=-2.572,64.710,59.508,-142.1219,1.6993,0.0000
C00666=0.000,64.758,59.526,-142.0985,-0.0006,0.0000
C00667=0.000,63.425,61.276,-142.4756,-0.0007,0.0000
C00668=2.450,63.381,61.257,-142.4979,-1.6531,0.0000
C00669=5.367,63.268,61.285,-142.6050,-0.9243,0.0000
C00670=8.682,63.886,61.945,-143.3805,2.7245,0.0000
C00671=10.270,66.465,63.612,-144.2096,4.9339,0.0000
C00672=11.189,70.924,65.929,-145.2247,7.0219,0.0000
C00673=12.084,76.878,68.324,-147.6714,10.3439,0.0000
C00674=13.063,83.550,70.157,-158.1723,15.5882,0.0000
C00675=14.270,89.726,71.060,-179.5273,1.4413,0.0000
C00676=17.683,94.235,71.535,179.2121,-3.0474,0.0000
C00677=22.929,96.378,71.920,178.8906,-4.5299,0.0000
C00678=28.946,95.684,72.309,178.8364,-4.7631,0.0000
C00679=35.156,93.612,72.565,178.8864,-4.5095,0.0000
C00680=41.335,91.053,72.565,-177.5931,3.9735,0.0000
C00681=47.191,88.127,72.309,-177.4481,4.1878,0.0000
C00682=51.936,84.362,71.920,-177.5756,3.9850,0.0000
C00683=54.130,79.138,71.535,-178.4005,2.7112,0.0000
C00684=53.356,73.536,71.060,179.3149,-1.3533,0.0000
C00685=49.842,68.316,70.157,-175.9552,-26.3120,0.0000
C00686=45.816,62.906,68.324,-163.5760,-29.9314,0.0000
C00687=42.239,58.063,65.929,-158.9450,-29.1254,0.0000
C00688=39.736,54.260,63.612,-156.5127,-28.2172,0.0000
C00689=39.035,51.313,61.945,-154.1919,-27.0599,0.0000
C00690=40.942,48.532,61.285,-150.9747,-24.7064,0.0000
C00691=43.085,46.550,61.257,-150.3884,-24.1986,0.0000
C00692=44.848,44.848,61.276,-151.4949,-25.5113,0.0000
C00693=46.550,43.085,61.257,-152.6661,-26.7891,0.0000
C00694=48.532,40.942,61.285,-152.2474,-26.1527,0.0000
C00695=51.313,39.035,61.945,-150.4274,-22.8111,0.0000
C00696=54.260,39.736,63.612,-149.6700,-20.5596,0.0000
C00697=58.063,42.239,65.929,-149.1613,-18.2906,0.0000
C00698=62.906,45.816,68.324,-149.0258,-14.1840,0.0000
C00699=68.316,49.842,70.157,-153.6307,-3.6258,0.0000
C00700=73.536,53.356,71.060,-178.6466,0.6849,0.0000
C00701=79.138,54.130,71.535,177.2877,-1.5977,0.0000
C00702=84.362,51.936,71.920,176.0115,-2.4186,0.0000
C00703=88.127,47.191,72.309,175.8081,-2.5451,0.0000
C00704=91.053,41.335,72.565,176.0230,-2.4011,0.0000
C00705=93.612,35.156,72.565,-175.4897,1.1102,0.0000
C00706=95.684,28.946,72.309,-175.2359,1.1596,0.0000
C00707=96.378,22.929,71.920,-175.4692,1.1059,0.0000
C00708=94.235,17.683,71.535,-176.9523,0.7868,0.0000
C00709=89.726,14.270,71.060,178.5586,-0.4726,0.0000
C00710=83.550,13.063,70.157,163.2729,-20.9860,0.0000
C00711=76.878,12.084,68.324,167.8111,-31.7412,0.0000
C00712=70.924,11.189,65.929,171.4718,-34.4774,0.0000
C00713=66.465,10.270,63.612,173.9253,-35.6375,0.0000
C00714=63.886,8.682,61.945,176.6069,-36.5714,0.0000
C00715=63.268,5.367,61.285,-178.8366,-37.3893,0.0000
C00716=63.381,2.450,61.257,-177.9166,-37.4838,0.0000
C00717=63.425,0.000,61.276,-179.9992,-37.5244,0.0000
C00718=63.381,-2.450,61.257,177.9157,-37.4838,0.0000
C00719=63.268,-5.367,61.285,178.8382,-37.3892,0.0000
C00720=63.886,-8.682,61.945,-176.6064,-36.5713,0.0000
C00721=66.465,-10.270,63.612,-173.9251,-35.6375,0.0000
C00722=70.924,-11.189,65.929,-171.4717,-34.4774,0.0000
C00723=76.878,-12.084,68.324,-167.8113,-31.7414,0.0000
C00724=83.550,-13.063,70.157,-163.2730,-20.9868,0.0000
C00725=89.726,-14.270,71.060,-178.5586,-0.4726,0.0000
C00726=94.235,-17.683,71.535,176.9523,0.7868,0.0000
C00727=96.378,-22.929,71.920,175.4692,1.1059,0.0000
C00728=95.684,-28.946,72.309,175.2359,1.1596,0.0000
C00729=93.612,-35.156,72.565,175.4897,1.1102,0.0000
C00730=91.053,-41.335,72.565,-176.0230,-2.4011,0.0000
C00731=88.127,-47.191,72.309,-175.8081,-2.5451,0.0000
C00732=84.362,-51.936,71.920,-176.0115,-2.4186,0.0000
C00733=79.138,-54.130,71.535,-177.2877,-1.5977,0.0000
C00734=73.536,-53.356,71.060,178.6466,0.6849,0.0000
C00735=68.316,-49.842,70.157,153.6312,-3.6251,0.0000
C00736=62.906,-45.816,68.324,149.0258,-14.1837,0.0000
C00737=58.063,-42.239,65.929,149.1614,-18.2906,0.0000
C00738=54.260,-39.736,63.612,149.6700,-20.5597,0.0000
C00739=51.313,-39.035,61.945,150.4276,-22.8115,0.0000
C00740=48.532,-40.942,61.285,152.2481,-26.1537,0.0000
C00741=46.550,-43.085,61.257,152.6656,-26.7886,0.0000
C00742=44.848,-44.848,61.276,151.4958,-25.5124,0.0000
C00743=43.085,-46.550,61.257,150.3880,-24.1981,0.0000
C00744=40.942,-48.532,61.285,150.9757,-24.7073,0.0000
C00745=39.035,-51.313,61.945,154.1923,-27.0602,0.0000
C00746=39.736,-54.260,63.612,156.5128,-28.2173,0.0000
C00747=42.239,-58.063,65.929,158.9450,-29.1254,0.0000
C00748=45.816,-62.906,68.324,163.5757,-29.9314,0.0000
C00749=49.842,-68.316,70.157,175.9545,-26.3124,0.0000
C00750=53.356,-73.536,71.060,-179.3149,-1.3533,0.0000
C00751=54.130,-79.138,71.535,178.4005,2.7112,0.0000
C00752=51.936,-84.362,71.920,177.5756,3.9850,0.0000
C00753=47.191,-88.127,72.309,177.4481,4.1878,0.0000
C00754=41.335,-91.053,72.565,177.5931,3.9735,0.0000
C00755=35.156,-93.612,72.565,-178.8864,-4.5095,0.0000
C00756=28.946,-95.684,72.309,-178.8364,-4.7631,0.0000
C00757=22.929,-96.378,71.920,-178.8906,-4.5299,0.0000
C00758=17.683,-94.235,71.535,-179.2121,-3.0474,0.0000
C00759=14.270,-89.726,71.060,179.5273,1.4413,0.0000
C00760=13.063,-83.550,70.157,158.1723,15.5882,0.0000
C00761=12.084,-76.878,68.324,147.6714,10.3439,0.0000
C00762=11.189,-70.924,65.929,145.2247,7.0219,0.0000
C00763=10.270,-66.465,63.612,144.2096,4.9339,0.0000
C00764=8.682,-63.886,61.945,143.3805,2.7245,0.0000
C00765=5.367,-63.268,61.285,142.6050,-0.9243,0.0000
C00766=2.450,-63.381,61.257,142.4979,-1.6531,0.0000
C00767=0.000,-63.425,61.276,142.4756,-0.0007,0.0000
C00768=0.000,-63.425,61.276,142.4756,-0.0007,0.0000
C00769=-2.450,-63.381,61.257,142.4979,1.6538,0.0000
C00770=-5.367,-63.268,61.285,142.6051,0.9231,0.0000
C00771=-8.682,-63.886,61.945,143.3806,-2.7249,0.0000
C00772=-10.270,-66.465,63.612,144.2096,-4.9340,0.0000
C00773=-11.189,-70.924,65.929,145.2247,-7.0219,0.0000
C00774=-12.084,-76.878,68.324,147.6712,-10.3437,0.0000
C00775=-13.063,-83.550,70.157,158.1715,-15.5881,0.0000
C00776=-14.270,-89.726,71.060,179.5273,-1.4413,0.0000
C00777=-17.683,-94.235,71.535,-179.2121,3.0474,0.0000
C00778=-22.929,-96.378,71.920,-178.8906,4.5299,0.0000
C00779=-28.946,-95.684,72.309,-178.8364,4.7631,0.0000
C00780=-35.156,-93.612,72.565,-178.8864,4.5095,0.0000
C00781=-41.335,-91.053,72.565,177.5931,-3.9735,0.0000
C00782=-47.191,-88.127,72.309,177.4481,-4.1878,0.0000
C00783=-51.936,-84.362,71.920,177.5756,-3.9850,0.0000
C00784=-54.130,-79.138,71.535,178.4005,-2.7112,0.0000
C00785=-53.356,-73.536,71.060,-179.3149,1.3533,0.0000
C00786=-49.842,-68.316,70.157,175.9552,26.3120,0.0000
C00787=-45.816,-62.906,68.324,163.5760,29.9314,0.0000
C00788=-42.239,-58.063,65.929,158.9450,29.1254,0.0000
C00789=-39.736,-54.260,63.612,156.5127,28.2172,0.0000
C00790=-39.035,-51.313,61.945,154.1919,27.0599,0.0000
C00791=-40.942,-48.532,61.285,150.9747,24.7064,0.0000
C00792=-43.085,-46.550,61.257,150.3884,24.1986,0.0000
C00793=-44.848,-44.848,61.276,151.4949,25.5113,0.0000
C00794=-46.550,-43.085,61.257,152.6661,26.7891,0.0000
C00795=-48.532,-40.942,61.285,152.2474,26.1527,0.0000
C00796=-51.313,-39.035,61.945,150.4274,22.8111,0.0000
C00797=-54.260,-39.736,63.612,149.6700,20.5596,0.0000
C00798=-58.063,-42.239,65.929,149.1613,18.2906,0.0000
C00799=-62.906,-45.816,68.324,149.0258,14.1840,0.0000
C00800=-68.316,-49.842,70.157,153.6307,3.6258,0.0000
C00801=-73.536,-53.356,71.060,178.6466,-0.6849,0.0000
C00802=-79.138,-54.130,71.535,-177.2877,1.5977,0.0000
C00803=-84.362,-51.936,71.920,-176.0115,2.4186,0.0000
C00804=-88.127,-47.191,72.309,-175.8081,2.5451,0.0000
C00805=-91.053,-41.335,72.565,-176.0230,2.4011,0.0000
C00806=-93.612,-35.156,72.565,175.4897,-1.1102,0.0000
C00807=-95.684,-28.946,72.309,175.2359,-1.1596,0.0000
C00808=-96.378,-22.929,71.920,175.4692,-1.1059,0.0000
C00809=-94.235,-17.683,71.535,176.9523,-0.7868,0.0000
C00810=-89.726,-14.270,71.060,-178.5586,0.4726,0.0000
C00811=-83.550,-13.063,70.157,-163.2729,20.9860,0.0000
C00812=-76.878,-12.084,68.324,-167.8111,31.7412,0.0000
C00813=-70.924,-11.189,65.929,-171.4718,34.4774,0.0000
C00814=-66.465,-10.270,63.612,-173.9253,35.6375,0.0000
C00815=-63.886,-8.682,61.945,-176.6069,36.5714,0.0000
C00816=-63.268,-5.367,61.285,178.8366,37.3893,0.0000
C00817=-63.381,-2.450,61.257,177.9166,37.4838,0.0000
C00818=-63.425,0.000,61.276,179.9992,37.5244,0.0000
C00819=-63.381,2.450,61.257,-177.9157,37.4838,0.0000
C00820=-63.268,5.367,61.285,-178.8382,37.3892,0.0000
C00821=-63.886,8.682,61.945,176.6064,36.5713,0.0000
C00822=-66.465,10.270,63.612,173.9251,35.6375,0.0000
C00823=-70.924,11.189,65.929,171.4717,34.4774,0.0000
C00824=-76.878,12.084,68.324,167.8113,31.7414,0.0000
C00825=-83.550,13.063,70.157,163.2730,20.9868,0.0000
C00826=-89.726,14.270,71.060,178.5586,0.4726,0.0000
C00827=-94.235,17.683,71.535,-176.9523,-0.7868,0.0000
C00828=-96.378,22.929,71.920,-175.4692,-1.1059,0.0000
C00829=-95.684,28.946,72.309,-175.2359,-1.1596,0.0000
C00830=-93.612,35.156,72.565,-175.4897,-1.1102,0.0000
C00831=-91.053,41.335,72.565,176.0230,2.4011,0.0000
C00832=-88.127,47.191,72.309,175.8081,2.5451,0.0000
C00833=-84.362,51.936,71.920,176.0115,2.4186,0.0000
C00834=-79.138,54.130,71.535,177.2877,1.5977,0.0000
C00835=-73.536,53.356,71.060,-178.6466,-0.6849,0.0000
C00836=-68.316,49.842,70.157,-153.6312,3.6251,0.0000
C00837=-62.906,45.816,68.324,-149.0258,14.1837,0.0000
C00838=-58.063,42.239,65.929,-149.1614,18.2906,0.0000
C00839=-54.260,39.736,63.612,-149.6700,20.5597,0.0000
C00840=-51.313,39.035,61.945,-150.4276,22.8115,0.0000
C00841=-48.532,40.942,61.285,-152.2481,26.1537,0.0000
C00842=-46.550,43.085,61.257,-152.6656,26.7886,0.0000
C00843=-44.848,44.848,61.276,-151.4958,25.5124,0.0000
C00844=-43.085,46.550,61.257,-150.3880,24.1981,0.0000
C00845=-40.942,48.532,61.285,-150.9757,24.7073,0.0000
C00846=-39.035,51.313,61.945,-154.1923,27.0602,0.0000
C00847=-39.736,54.260,63.612,-156.5128,28.2173,0.0000
C00848=-42.239,58.063,65.929,-158.9450,29.1254,0.0000
C00849=-45.816,62.906,68.324,-163.5757,29.9314,0.0000
C00850=-49.842,68.316,70.157,-175.9545,26.3124,0.0000
C00851=-53.356,73.536,71.060,179.3149,1.3533,0.0000
C00852=-54.130,79.138,71.535,-178.4005,-2.7112,0.0000
C00853=-51.936,84.362,71.920,-177.5756,-3.9850,0.0000
C00854=-47.191,88.127,72.309,-177.4481,-4.1878,0.0000
C00855=-41.335,91.053,72.565,-177.5931,-3.9735,0.0000
C00856=-35.156,93.612,72.565,178.8864,4.5095,0.0000
C00857=-28.946,95.684,72.309,178.8364,4.7631,0.0000
C00858=-22.929,96.378,71.920,178.8906,4.5299,0.0000
C00859=-17.683,94.235,71.535,179.2121,3.0474,0.0000
C00860=-14.270,89.726,71.060,-179.5273,-1.4413,0.0000
C00861=-13.063,83.550,70.157,-158.1715,-15.5881,0.0000
C00862=-12.084,76.878,68.324,-147.6712,-10.3437,0.0000
C00863=-11.189,70.924,65.929,-145.2247,-7.0219,0.0000
C00864=-10.270,66.465,63.612,-144.2096,-4.9340,0.0000
C00865=-8.682,63.886,61.945,-143.3806,-2.7249,0.0000
C00866=-5.367,63.268,61.285,-142.6051,0.9231,0.0000
C00867=-2.450,63.381,61.257,-142.4979,1.6538,0.0000
C00868=0.000,63.425,61.276,-142.4756,-0.0007,0.0000
C00869=0.000,62.111,63.041,-142.8998,-0.0007,0.0000
C00870=2.330,62.072,63.021,-142.9209,-1.6044,0.0000
C00871=5.165,61.970,63.050,-143.0255,-0.8915,0.0000
C00872=8.436,62.639,63.741,-143.7971,2.7451,0.0000
C00873=9.975,65.350,65.485,-144.6127,4.9284,0.0000
C00874=10.861,70.011,67.904,-145.6424,7.0639,0.0000
C00875=11.743,76.212,70.393,-148.3348,10.6221,0.0000
C00876=12.712,83.133,72.289,-162.2488,15.5790,0.0000
C00877=13.898,89.524,73.219,179.8928,-0.3726,0.0000
C00878=17.338,94.193,73.707,179.0724,-3.8680,0.0000
C00879=22.659,96.427,74.103,178.8239,-5.0916,0.0000
C00880=28.778,95.739,74.502,178.7817,-5.2678,0.0000
C00881=35.099,93.634,74.765,178.8286,-5.0120,0.0000
C00882=41.391,91.028,74.765,-177.2766,4.3688,0.0000
C00883=47.349,88.047,74.502,-177.1277,4.5823,0.0000
C00884=52.162,84.206,74.103,-177.2233,4.4283,0.0000
C00885=54.344,78.865,73.707,-177.9172,3.3893,0.0000
C00886=53.475,73.130,73.219,-179.8124,0.3393,0.0000
C00887=49.795,67.773,72.289,-178.8909,-23.4264,0.0000
C00888=45.586,62.194,70.393,-164.3409,-29.6816,0.0000
C00889=41.825,57.185,67.904,-159.3306,-28.8808,0.0000
C00890=39.156,53.262,65.485,-156.8538,-27.9512,0.0000
C00891=38.328,50.258,63.741,-154.5660,-26.8102,0.0000
C00892=40.167,47.472,63.050,-151.3600,-24.4716,0.0000
C00893=42.244,45.539,63.021,-150.7861,-23.9765,0.0000
C00894=43.919,43.919,63.041,-151.8623,-25.2473,0.0000
C00895=45.539,42.244,63.021,-152.9994,-26.4852,0.0000
C00896=47.472,40.167,63.050,-152.5890,-25.8636,0.0000
C00897=50.258,38.328,63.741,-150.7686,-22.5382,0.0000
C00898=53.262,39.156,65.485,-150.0120,-20.3175,0.0000
C00899=57.185,41.825,67.904,-149.4790,-18.0035,0.0000
C00900=62.194,45.586,70.393,-149.3773,-13.5623,0.0000
C00901=67.773,49.795,72.289,-156.5690,-1.0182,0.0000
C00902=73.130,53.475,73.219,179.6607,-0.1876,0.0000
C00903=78.865,54.344,73.707,176.6084,-2.0791,0.0000
C00904=84.206,52.162,74.103,175.5665,-2.7684,0.0000
C00905=88.047,47.349,74.502,175.4119,-2.8631,0.0000
C00906=91.028,41.391,74.765,175.6263,-2.7154,0.0000
C00907=93.634,35.099,74.765,-174.9870,1.1669,0.0000
C00908=95.739,28.778,74.502,-174.7310,1.2131,0.0000
C00909=96.427,22.659,74.103,-174.9073,1.1715,0.0000
C00910=94.193,17.338,73.707,-176.1315,0.9254,0.0000
C00911=89.524,13.898,73.219,-179.6274,0.1072,0.0000
C00912=83.133,12.712,72.289,163.6827,-17.0786,0.0000
C00913=76.212,11.743,70.393,167.5737,-31.0616,0.0000
C00914=70.011,10.861,67.904,171.4634,-34.0609,0.0000
C00915=65.350,9.975,65.485,173.9623,-35.2370,0.0000
C00916=62.639,8.436,63.741,176.5995,-36.1548,0.0000
C00917=61.970,5.165,63.050,-178.8841,-36.9692,0.0000
C00918=62.072,2.330,63.021,-177.9893,-37.0621,0.0000
C00919=62.111,0.000,63.041,-179.9991,-37.1002,0.0000
C00920=62.072,-2.330,63.021,177.9883,-37.0621,0.0000
C00921=61.970,-5.165,63.050,178.8857,-36.9692,0.0000
C00922=62.640,-8.436,63.741,-176.5990,-36.1547,0.0000
C00923=65.350,-9.975,65.485,-173.9622,-35.2370,0.0000
C00924=70.011,-10.861,67.904,-171.4634,-34.0609,0.0000
C00925=76.212,-11.743,70.393,-167.5739,-31.0618,0.0000
C00926=83.133,-12.712,72.289,-163.6826,-17.0795,0.0000
C00927=89.524,-13.898,73.219,179.6274,0.1072,0.0000
C00928=94.193,-17.338,73.707,176.1315,0.9254,0.0000
C00929=96.427,-22.659,74.103,174.9073,1.1715,0.0000
C00930=95.739,-28.778,74.502,174.7310,1.2131,0.0000
C00931=93.634,-35.099,74.765,174.9870,1.1669,0.0000
C00932=91.028,-41.391,74.765,-175.6263,-2.7154,0.0000
C00933=88.047,-47.349,74.502,-175.4119,-2.8631,0.0000
C00934=84.206,-52.162,74.103,-175.5665,-2.7684,0.0000
C00935=78.865,-54.344,73.707,-176.6084,-2.0791,0.0000
C00936=73.130,-53.475,73.219,-179.6607,-0.1876,0.0000
C00937=67.773,-49.795,72.289,156.5697,-1.0177,0.0000
C00938=62.194,-45.586,70.393,149.3773,-13.5620,0.0000
C00939=57.185,-41.825,67.904,149.4790,-18.0035,0.0000
C00940=53.262,-39.156,65.485,150.0121,-20.3176,0.0000
C00941=50.258,-38.328,63.741,150.7688,-22.5386,0.0000
C00942=47.472,-40.167,63.050,152.5898,-25.8646,0.0000
C00943=45.539,-42.244,63.021,152.9989,-26.4846,0.0000
C00944=43.919,-43.919,63.041,151.8633,-25.2484,0.0000
C00945=42.244,-45.539,63.021,150.7856,-23.9759,0.0000
C00946=40.167,-47.472,63.050,151.3610,-24.4725,0.0000
C00947=38.328,-50.258,63.741,154.5663,-26.8104,0.0000
C00948=39.156,-53.262,65.485,156.8539,-27.9513,0.0000
C00949=41.825,-57.185,67.904,159.3306,-28.8808,0.0000
C00950=45.586,-62.194,70.393,164.3406,-29.6816,0.0000
C00951=49.795,-67.773,72.289,178.8903,-23.4270,0.0000
C00952=53.475,-73.130,73.219,179.8124,0.3393,0.0000
C00953=54.344,-78.865,73.707,177.9172,3.3893,0.0000
C00954=52.162,-84.206,74.103,177.2233,4.4283,0.0000
C00955=47.349,-88.047,74.502,177.1277,4.5823,0.0000
C00956=41.391,-91.028,74.765,177.2766,4.3688,0.0000
C00957=35.099,-93.634,74.765,-178.8286,-5.0120,0.0000
C00958=28.778,-95.739,74.502,-178.7817,-5.2678,0.0000
C00959=22.659,-96.427,74.103,-178.8239,-5.0916,0.0000
C00960=17.338,-94.193,73.707,-179.0724,-3.8680,0.0000
C00961=13.898,-89.524,73.219,-179.8928,-0.3726,0.0000
C00962=12.712,-83.133,72.289,162.2488,15.5790,0.0000
C00963=11.743,-76.212,70.393,148.3348,10.6221,0.0000
C00964=10.861,-70.011,67.904,145.6424,7.0639,0.0000
C00965=9.975,-65.350,65.485,144.6127,4.9284,0.0000
C00966=8.436,-62.639,63.741,143.7971,2.7451,0.0000
C00967=5.165,-61.970,63.050,143.0255,-0.8915,0.0000
C00968=2.330,-62.072,63.021,142.9209,-1.6044,0.0000
C00969=0.000,-62.111,63.041,142.8998,-0.0007,0.0000
C00970=0.000,-62.111,63.041,142.8998,-0.0007,0.0000
C00971=-2.330,-62.072,63.021,142.9209,1.6051,0.0000
C00972=-5.165,-61.970,63.050,143.0256,0.8903,0.0000
C00973=-8.436,-62.640,63.741,143.7972,-2.7455,0.0000
C00974=-9.975,-65.350,65.485,144.6127,-4.9285,0.0000
C00975=-10.861,-70.011,67.904,145.6423,-7.0639,0.0000
C00976=-11.743,-76.212,70.393,148.3346,-10.6218,0.0000
C00977=-12.712,-83.133,72.289,162.2479,-15.5790,0.0000
C00978=-13.898,-89.524,73.219,-179.8928,0.3726,0.0000
C00979=-17.338,-94.193,73.707,-179.0724,3.8680,0.0000
C00980=-22.659,-96.427,74.103,-178.8239,5.0916,0.0000
C00981=-28.778,-95.739,74.502,-178.7817,5.2678,0.0000
C00982=-35.099,-93.634,74.765,-178.8286,5.0120,0.0000
C00983=-41.391,-91.028,74.765,177.2766,-4.3688,0.0000
C00984=-47.349,-88.047,74.502,177.1277,-4.5823,0.0000
C00985=-52.162,-84.206,74.103,177.2233,-4.4283,0.0000
C00986=-54.344,-78.865,73.707,177.9172,-3.3893,0.0000
C00987=-53.475,-73.130,73.219,179.8124,-0.3393,0.0000
C00988=-49.795,-67.773,72.289,178.8909,23.4264,0.0000
C00989=-45.586,-62.194,70.393,164.3409,29.6816,0.0000
C00990=-41.825,-57.185,67.904,159.3306,28.8808,0.0000
C00991=-39.156,-53.262,65.485,156.8538,27.9512,0.0000
C00992=-38.328,-50.258,63.741,154.5660,26.8102,0.0000
C00993=-40.167,-47.472,63.050,151.3600,24.4716,0.0000
C00994=-42.244,-45.539,63.021,150.7861,23.9765,0.0000
C00995=-43.919,-43.919,63.041,151.8623,25.2473,0.0000
C00996=-45.539,-42.244,63.021,152.9994,26.4852,0.0000
C00997=-47.472,-40.167,63.050,152.5890,25.8636,0.0000
C00998=-50.258,-38.328,63.741,150.7686,22.5382,0.0000
C00999=-53.262,-39.156,65.485,150.0120,20.3175,0.0000
C01000=-57.185,-41.825,67.904,149.4790,18.0035,0.0000
C01001=-62.194,-45.586,70.393,149.3773,13.5623,0.0000
C01002=-67.773,-49.795,72.289,156.5690,1.0182,0.0000
C01003=-73.130,-53.475,73.219,-179.6607,0.1876,0.0000
C01004=-78.865,-54.344,73.707,-176.6084,2.0791,0.0000
C01005=-84.206,-52.162,74.103,-175.5665,2.7684,0.0000
C01006=-88.047,-47.349,74.502,-175.4119,2.8631,0.0000
C01007=-91.028,-41.391,74.765,-175.6263,2.7154,0.0000
C01008=-93.634,-35.099,74.765,174.9870,-1.1669,0.0000
C01009=-95.739,-28.778,74.502,174.7310,-1.2131,0.0000
C01010=-96.427,-22.659,74.103,174.9073,-1.1715,0.0000
C01011=-94.193,-17.338,73.707,176.1315,-0.9254,0.0000
C01012=-89.524,-13.898,73.219,179.6274,-0.1072,0.0000
C01013=-83.133,-12.712,72.289,-163.6827,17.0786,0.0000
C01014=-76.212,-11.743,70.393,-167.5737,31.0616,0.0000
C01015=-70.011,-10.861,67.904,-171.4634,34.0609,0.0000
C01016=-65.350,-9.975,65.485,-173.9623,35.2370,0.0000
C01017=-62.639,-8.436,63.741,-176.5995,36.1548,0.0000
C01018=-61.970,-5.165,63.050,178.8841,36.9692,0.0000
C01019=-62.072,-2.330,63.021,177.9893,37.0621,0.0000
C01020=-62.111,0.000,63.041,179.9991,37.1002,0.0000
C01021=-62.072,2.330,63.021,-177.9883,37.0621,0.0000
C01022=-61.970,5.165,63.050,-178.8857,36.9692,0.0000
C01023=-62.640,8.436,63.741,176.5990,36.1547,0.0000
C01024=-65.350,9.975,65.485,173.9622,35.2370,0.0000
C01025=-70.011,10.861,67.904,171.4634,34.0609,0.0000
C01026=-76.212,11.743,70.393,167.5739,31.0618,0.0000
C01027=-83.133,12.712,72.289,163.6826,17.0795,0.0000
C01028=-89.524,13.898,73.219,-179.6274,-0.1072,0.0000
C01029=-94.193,17.338,73.707,-176.1315,-0.9254,0.0000
C01030=-96.427,22.659,74.103,-174.9073,-1.1715,0.0000
C01031=-95.739,28.778,74.502,-174.7310,-1.2131,0.0000
C01032=-93.634,35.099,74.765,-174.9870,-1.1669,0.0000
C01033=-91.028,41.391,74.765,175.6263,2.7154,0.0000
C01034=-88.047,47.349,74.502,175.4119,2.8631,0.0000
C01035=-84.206,52.162,74.103,175.5665,2.7684,0.0000
C01036=-78.865,54.344,73.707,176.6084,2.0791,0.0000
C01037=-73.130,53.475,73.219,179.6607,0.1876,0.0000
C01038=-67.773,49.795,72.289,-156.5697,1.0177,0.0000
C01039=-62.194,45.586,70.393,-149.3773,13.5620,0.0000
C01040=-57.185,41.825,67.904,-149.4790,18.0035,0.0000
C01041=-53.262,39.156,65.485,-150.0121,20.3176,0.0000
C01042=-50.258,38.328,63.741,-150.7688,22.5386,0.0000
C01043=-47.472,40.167,63.050,-152.5898,25.8646,0.0000
C01044=-45.539,42.244,63.021,-152.9989,26.4846,0.0000
C01045=-43.919,43.919,63.041,-151.8633,25.2484,0.0000
C01046=-42.244,45.539,63.021,-150.7856,23.9759,0.0000
C01047=-40.167,47.472,63.050,-151.3610,24.4725,0.0000
C01048=-38.328,50.258,63.741,-154.5663,26.8104,0.0000
C01049=-39.156,53.262,65.485,-156.8539,27.9513,0.0000
C01050=-41.825,57.185,67.904,-159.3306,28.8808,0.0000
C01051=-45.586,62.194,70.393,-164.3406,29.6816,0.0000
C01052=-49.795,67.773,72.289,-178.8903,23.4270,0.0000
C01053=-53.475,73.130,73.219,-179.8124,-0.3393,0.0000
C01054=-54.344,78.865,73.707,-177.9172,-3.3893,0.0000
C01055=-52.162,84.206,74.103,-177.2233,-4.4283,0.0000
C01056=-47.349,88.047,74.502,-177.1277,-4.5823,0.0000
C01057=-41.391,91.028,74.765,-177.2766,-4.3688,0.0000
C01058=-35.099,93.634,74.765,178.8286,5.0120,0.0000
C01059=-28.778,95.739,74.502,178.7817,5.2678,0.0000
C01060=-22.659,96.427,74.103,178.8239,5.0916,0.0000
C01061=-17.338,94.193,73.707,179.0724,3.8680,0.0000
C01062=-13.898,89.524,73.219,179.8928,0.3726,0.0000
C01063=-12.712,83.133,72.289,-162.2479,-15.5790,0.0000
C01064=-11.743,76.212,70.393,-148.3346,-10.6218,0.0000
C01065=-10.861,70.011,67.904,-145.6423,-7.0639,0.0000
C01066=-9.975,65.350,65.485,-144.6127,-4.9285,0.0000
C01067=-8.436,62.640,63.741,-143.7972,-2.7455,0.0000
C01068=-5.165,61.970,63.050,-143.0256,0.8903,0.0000
C01069=-2.330,62.072,63.021,-142.9209,1.6051,0.0000
C01070=0.000,62.111,63.041,-142.8998,-0.0007,0.0000
C01071=0.000,60.820,64.822,-143.3720,-0.0008,0.0000
C01072=2.212,60.785,64.801,-143.3919,-1.5525,0.0000
C01073=4.967,60.695,64.832,-143.4939,-0.8622,0.0000
C01074=8.195,61.417,65.554,-144.2608,2.7560,0.0000
C01075=9.686,64.262,67.375,-145.0647,4.9141,0.0000
C01076=10.544,69.129,69.894,-146.1170,7.1061,0.0000
C01077=11.418,75.576,72.474,-149.1249,10.9344,0.0000
C01078=12.382,82.740,74.428,-168.4179,13.9743,0.0000
C01079=13.550,89.334,75.383,179.5556,-1.7205,0.0000
C01080=17.016,94.154,75.883,178.9906,-4.4951,0.0000
C01081=22.407,96.473,76.288,178.7889,-5.5267,0.0000
C01082=28.621,95.791,76.696,178.7540,-5.6654,0.0000
C01083=35.046,93.654,76.964,178.7968,-5.4173,0.0000
C01084=41.442,91.005,76.964,-177.0107,4.6770,0.0000
C01085=47.497,87.973,76.696,-176.8643,4.8821,0.0000
C01086=52.372,84.060,76.288,-176.9384,4.7597,0.0000
C01087=54.545,78.609,75.883,-177.5298,3.8897,0.0000
C01088=53.588,72.750,75.383,-179.0974,1.5307,0.0000
C01089=49.751,67.261,74.428,178.0124,-17.9702,0.0000
C01090=45.367,61.514,72.474,-165.2320,-29.3671,0.0000
C01091=41.426,56.337,69.894,-159.7627,-28.5978,0.0000
C01092=38.591,52.289,67.375,-157.2287,-27.6462,0.0000
C01093=37.634,49.223,65.554,-154.9718,-26.5219,0.0000
C01094=39.406,46.429,64.832,-151.7826,-24.2033,0.0000
C01095=41.417,44.545,64.801,-151.2256,-23.7259,0.0000
C01096=43.006,43.006,64.822,-152.2695,-24.9522,0.0000
C01097=44.545,41.417,64.801,-153.3703,-26.1478,0.0000
C01098=46.430,39.405,64.832,-152.9726,-25.5463,0.0000
C01099=49.223,37.634,65.554,-151.1548,-22.2431,0.0000
C01100=52.289,38.591,67.375,-150.3993,-20.0514,0.0000
C01101=56.337,41.426,69.894,-149.8418,-17.6805,0.0000
C01102=61.514,45.367,72.474,-149.8031,-12.8356,0.0000
C01103=67.261,49.751,74.428,-162.0190,1.8903,0.0000
C01104=72.750,53.588,75.383,178.4692,-0.9023,0.0000
C01105=78.609,54.545,75.883,176.1066,-2.4645,0.0000
C01106=84.060,52.372,76.288,175.2335,-3.0510,0.0000
C01107=87.973,47.497,76.696,175.1106,-3.1244,0.0000
C01108=91.005,41.442,76.964,175.3166,-2.9793,0.0000
C01109=93.654,35.046,76.964,-174.5815,1.1978,0.0000
C01110=95.791,28.621,76.696,-174.3333,1.2399,0.0000
C01111=96.473,22.407,76.288,-174.4721,1.2055,0.0000
C01112=94.154,17.016,75.883,-175.5042,1.0063,0.0000
C01113=89.334,13.550,75.383,-178.2795,0.4442,0.0000
C01114=82.740,12.382,74.428,165.7470,-11.2348,0.0000
C01115=75.576,11.418,72.474,167.3147,-30.2551,0.0000
C01116=69.129,10.544,69.894,171.4599,-33.5880,0.0000
C01117=64.262,9.686,67.375,174.0128,-34.7883,0.0000
C01118=61.417,8.195,65.554,176.6060,-35.6916,0.0000
C01119=60.695,4.967,64.832,-178.9274,-36.5013,0.0000
C01120=60.785,2.212,64.801,-178.0662,-36.5924,0.0000
C01121=60.820,0.000,64.822,-179.9990,-36.6280,0.0000
C01122=60.785,-2.212,64.801,178.0652,-36.5924,0.0000
C01123=60.695,-4.967,64.832,178.9290,-36.5012,0.0000
C01124=61.417,-8.195,65.554,-176.6055,-35.6915,0.0000
C01125=64.262,-9.686,67.375,-174.0127,-34.7883,0.0000
C01126=69.129,-10.544,69.894,-171.4599,-33.5880,0.0000
C01127=75.576,-11.418,72.474,-167.3149,-30.2554,0.0000
C01128=82.740,-12.382,74.428,-165.7467,-11.2355,0.0000
C01129=89.334,-13.550,75.383,178.2795,0.4442,0.0000
C01130=94.154,-17.016,75.883,175.5042,1.0063,0.0000
C01131=96.473,-22.407,76.288,174.4721,1.2055,0.0000
C01132=95.791,-28.621,76.696,174.3333,1.2399,0.0000
C01133=93.654,-35.046,76.964,174.5815,1.1978,0.0000
C01134=91.005,-41.442,76.964,-175.3166,-2.9793,0.0000
C01135=87.973,-47.497,76.696,-175.1106,-3.1244,0.0000
C01136=84.060,-52.372,76.288,-175.2335,-3.0510,0.0000
C01137=78.609,-54.545,75.883,-176.1066,-2.4645,0.0000
C01138=72.750,-53.588,75.383,-178.4692,-0.9023,0.0000
C01139=67.261,-49.751,74.428,162.0197,1.8906,0.0000
C01140=61.514,-45.367,72.474,149.8032,-12.8353,0.0000
C01141=56.337,-41.426,69.894,149.8419,-17.6805,0.0000
C01142=52.289,-38.591,67.375,150.3994,-20.0515,0.0000
C01143=49.223,-37.634,65.554,151.1550,-22.2434,0.0000
C01144=46.429,-39.406,64.832,152.9734,-25.5473,0.0000
C01145=44.545,-41.417,64.801,153.3697,-26.1471,0.0000
C01146=43.006,-43.006,64.822,152.2706,-24.9534,0.0000
C01147=41.417,-44.545,64.801,151.2250,-23.7253,0.0000
C01148=39.405,-46.430,64.832,151.7835,-24.2043,0.0000
C01149=37.634,-49.223,65.554,154.9722,-26.5222,0.0000
C01150=38.591,-52.289,67.375,157.2287,-27.6463,0.0000
C01151=41.426,-56.337,69.894,159.7626,-28.5978,0.0000
C01152=45.367,-61.514,72.474,165.2316,-29.3672,0.0000
C01153=49.751,-67.261,74.428,-178.0127,-17.9709,0.0000
C01154=53.588,-72.750,75.383,179.0974,1.5307,0.0000
C01155=54.545,-78.609,75.883,177.5298,3.8897,0.0000
C01156=52.372,-84.060,76.288,176.9384,4.7597,0.0000
C01157=47.497,-87.973,76.696,176.8643,4.8821,0.0000
C01158=41.442,-91.005,76.964,177.0107,4.6770,0.0000
C01159=35.046,-93.654,76.964,-178.7968,-5.4173,0.0000
C01160=28.621,-95.791,76.696,-178.7540,-5.6654,0.0000
C01161=22.407,-96.473,76.288,-178.7889,-5.5267,0.0000
C01162=17.016,-94.154,75.883,-178.9906,-4.4951,0.0000
C01163=13.550,-89.334,75.383,-179.5556,-1.7205,0.0000
C01164=12.382,-82.740,74.428,168.4179,13.9743,0.0000
C01165=11.418,-75.576,72.474,149.1249,10.9344,0.0000
C01166=10.544,-69.129,69.894,146.1170,7.1061,0.0000
C01167=9.686,-64.262,67.375,145.0647,4.9141,0.0000
C01168=8.195,-61.417,65.554,144.2608,2.7560,0.0000
C01169=4.967,-60.695,64.832,143.4939,-0.8622,0.0000
C01170=2.212,-60.785,64.801,143.3919,-1.5525,0.0000
C01171=0.000,-60.820,64.822,143.3720,-0.0008,0.0000
C01172=0.000,-60.820,64.822,143.3720,-0.0008,0.0000
C01173=-2.212,-60.785,64.801,143.3919,1.5534,0.0000
C01174=-4.967,-60.695,64.832,143.4940,0.8609,0.0000
C01175=-8.195,-61.417,65.554,144.2608,-2.7564,0.0000
C01176=-9.686,-64.262,67.375,145.0647,-4.9143,0.0000
C01177=-10.544,-69.129,69.894,146.1169,-7.1061,0.0000
C01178=-11.418,-75.576,72.474,149.1247,-10.9342,0.0000
C01179=-12.382,-82.740,74.428,168.4172,-13.9746,0.0000
C01180=-13.550,-89.334,75.383,-179.5556,1.7205,0.0000
C01181=-17.016,-94.154,75.883,-178.9906,4.4951,0.0000
C01182=-22.407,-96.473,76.288,-178.7889,5.5267,0.0000
C01183=-28.621,-95.791,76.696,-178.7540,5.6654,0.0000
C01184=-35.046,-93.654,76.964,-178.7968,5.4173,0.0000
C01185=-41.442,-91.005,76.964,177.0107,-4.6770,0.0000
C01186=-47.497,-87.973,76.696,176.8643,-4.8821,0.0000
C01187=-52.372,-84.060,76.288,176.9384,-4.7597,0.0000
C01188=-54.545,-78.609,75.883,177.5298,-3.8897,0.0000
C01189=-53.588,-72.750,75.383,179.0974,-1.5307,0.0000
C01190=-49.751,-67.261,74.428,-178.0124,17.9702,0.0000
C01191=-45.367,-61.514,72.474,165.2320,29.3671,0.0000
C01192=-41.426,-56.337,69.894,159.7627,28.5978,0.0000
C01193=-38.591,-52.289,67.375,157.2287,27.6462,0.0000
C01194=-37.634,-49.223,65.554,154.9718,26.5219,0.0000
C01195=-39.406,-46.429,64.832,151.7826,24.2033,0.0000
C01196=-41.417,-44.545,64.801,151.2256,23.7259,0.0000
C01197=-43.006,-43.006,64.822,152.2695,24.9522,0.0000
C01198=-44.545,-41.417,64.801,153.3703,26.1478,0.0000
C01199=-46.430,-39.405,64.832,152.9726,25.5463,0.0000
C01200=-49.223,-37.634,65.554,151.1548,22.2431,0.0000
C01201=-52.289,-38.591,67.375,150.3993,20.0514,0.0000
C01202=-56.337,-41.426,69.894,149.8418,17.6805,0.0000
C01203=-61.514,-45.367,72.474,149.8031,12.8356,0.0000
C01204=-67.261,-49.751,74.428,162.0190,-1.8903,0.0000
C01205=-72.750,-53.588,75.383,-178.4692,0.9023,0.0000
C01206=-78.609,-54.545,75.883,-176.1066,2.4645,0.0000
C01207=-84.060,-52.372,76.288,-175.2335,3.0510,0.0000
C01208=-87.973,-47.497,76.696,-175.1106,3.1244,0.0000
C01209=-91.005,-41.442,76.964,-175.3166,2.9793,0.0000
C01210=-93.654,-35.046,76.964,174.5815,-1.1978,0.0000
C01211=-95.791,-28.621,76.696,174.3333,-1.2399,0.0000
C01212=-96.473,-22.407,76.288,174.4721,-1.2055,0.0000
C01213=-94.154,-17.016,75.883,175.5042,-1.0063,0.0000
C01214=-89.334,-13.550,75.383,178.2795,-0.4442,0.0000
C01215=-82.740,-12.382,74.428,-165.7470,11.2348,0.0000
C01216=-75.576,-11.418,72.474,-167.3147,30.2551,0.0000
C01217=-69.129,-10.544,69.894,-171.4599,33.5880,0.0000
C01218=-64.262,-9.686,67.375,-174.0128,34.7883,0.0000
C01219=-61.417,-8.195,65.554,-176.6060,35.6916,0.0000
C01220=-60.695,-4.967,64.832,178.9274,36.5013,0.0000
C01221=-60.785,-2.212,64.801,178.0662,36.5924,0.0000
C01222=-60.820,0.000,64.822,179.9990,36.6280,0.0000
C01223=-60.785,2.212,64.801,-178.0652,36.5924,0.0000
C01224=-60.695,4.967,64.832,-178.9290,36.5012,0.0000
C01225=-61.417,8.195,65.554,176.6055,35.6915,0.0000
C01226=-64.262,9.686,67.375,174.0127,34.7883,0.0000
C01227=-69.129,10.544,69.894,171.4599,33.5880,0.0000
C01228=-75.576,11.418,72.474,167.3149,30.2554,0.0000
C01229=-82.740,12.382,74.428,165.7467,11.2355,0.0000
C01230=-89.334,13.550,75.383,-178.2795,-0.4442,0.0000
C01231=-94.154,17.016,75.883,-175.5042,-1.0063,0.0000
C01232=-96.473,22.407,76.288,-174.4721,-1.2055,0.0000
C01233=-95.791,28.621,76.696,-174.3333,-1.2399,0.0000
C01234=-93.654,35.046,76.964,-174.5815,-1.1978,0.0000
C01235=-91.005,41.442,76.964,175.3166,2.9793,0.0000
C01236=-87.973,47.497,76.696,175.1106,3.1244,0.0000
C01237=-84.060,52.372,76.288,175.2335,3.0510,0.0000
C01238=-78.609,54.545,75.883,176.1066,2.4645,0.0000
C01239=-72.750,53.588,75.383,178.4692,0.9023,0.0000
C01240=-67.261,49.751,74.428,-162.0197,-1.8906,0.0000
C01241=-61.514,45.367,72.474,-149.8032,12.8353,0.0000
C01242=-56.337,41.426,69.894,-149.8419,17.6805,0.0000
C01243=-52.289,38.591,67.375,-150.3994,20.0515,0.0000
C01244=-49.223,37.634,65.554,-151.1550,22.2434,0.0000
C01245=-46.429,39.406,64.832,-152.9734,25.5473,0.0000
C01246=-44.545,41.417,64.801,-153.3697,26.1471,0.0000
C01247=-43.006,43.006,64.822,-152.2706,24.9534,0.0000
C01248=-41.417,44.545,64.801,-151.2250,23.7253,0.0000
C01249=-39.405,46.430,64.832,-151.7835,24.2043,0.0000
C01250=-37.634,49.223,65.554,-154.9722,26.5222,0.0000
C01251=-38.591,52.289,67.375,-157.2287,27.6463,0.0000
C01252=-41.426,56.337,69.894,-159.7626,28.5978,0.0000
C01253=-45.367,61.514,72.474,-165.2316,29.3672,0.0000
C01254=-49.751,67.261,74.428,178.0127,17.9709,0.0000
C01255=-53.588,72.750,75.383,-179.0974,-1.5307,0.0000
C01256=-54.545,78.609,75.883,-177.5298,-3.8897,0.0000
C01257=-52.372,84.060,76.288,-176.9384,-4.7597,0.0000
C01258=-47.497,87.973,76.696,-176.8643,-4.8821,0.0000
C01259=-41.442,91.005,76.964,-177.0107,-4.6770,0.0000
C01260=-35.046,93.654,76.964,178.7968,5.4173,0.0000
C01261=-28.621,95.791,76.696,178.7540,5.6654,0.0000
C01262=-22.407,96.473,76.288,178.7889,5.5267,0.0000
C01263=-17.016,94.154,75.883,178.9906,4.4951,0.0000
C01264=-13.550,89.334,75.383,179.5556,1.7205,0.0000
C01265=-12.382,82.740,74.428,-168.4172,-13.9746,0.0000
C01266=-11.418,75.576,72.474,-149.1247,-10.9342,0.0000
C01267=-10.544,69.129,69.894,-146.1169,-7.1061,0.0000
C01268=-9.686,64.262,67.375,-145.0647,-4.9142,0.0000
C01269=-8.195,61.417,65.554,-144.2608,-2.7564,0.0000
C01270=-4.967,60.695,64.832,-143.4940,0.8609,0.0000
C01271=-2.212,60.785,64.801,-143.3919,1.5534,0.0000
C01272=0.000,60.820,64.822,-143.3720,-0.0008,0.0000
C01273=0.000,59.554,66.621,-143.8937,-0.0009,0.0000
C01274=2.097,59.523,66.599,-143.9122,-1.4976,0.0000
C01275=4.772,59.445,66.632,-144.0113,-0.8357,0.0000
C01276=7.959,60.221,67.386,-144.7730,2.7581,0.0000
C01277=9.406,63.206,69.285,-145.5678,4.8928,0.0000
C01278=10.239,68.282,71.901,-146.6530,7.1518,0.0000
C01279=11.109,74.974,74.567,-150.0710,11.2878,0.0000
C01280=12.073,82.372,76.575,-176.8007,7.1331,0.0000
C01281=13.226,89.158,77.551,179.3588,-2.7181,0.0000
C01282=16.717,94.118,78.062,178.9478,-4.9659,0.0000
C01283=22.174,96.515,78.476,178.7775,-5.8532,0.0000
C01284=28.477,95.839,78.891,178.7470,-5.9677,0.0000
C01285=34.998,93.673,79.163,178.7855,-5.7335,0.0000
C01286=41.489,90.984,79.163,-176.7935,4.9078,0.0000
C01287=47.632,87.904,78.891,-176.6538,5.1000,0.0000
C01288=52.567,83.926,78.476,-176.7139,4.9979,0.0000
C01289=54.731,78.373,78.062,-177.2254,4.2522,0.0000
C01290=53.692,72.396,77.551,-178.5302,2.3748,0.0000
C01291=49.709,66.782,76.575,177.1888,-7.2941,0.0000
C01292=45.159,60.870,74.567,-166.2756,-28.9717,0.0000
C01293=41.042,55.523,71.901,-160.2467,-28.2755,0.0000
C01294=38.042,51.344,69.285,-157.6396,-27.3016,0.0000
C01295=36.955,48.211,67.386,-155.4109,-26.1948,0.0000
C01296=38.660,45.408,66.632,-152.2432,-23.9010,0.0000
C01297=40.607,43.572,66.599,-151.7075,-23.4457,0.0000
C01298=42.111,42.111,66.621,-152.7169,-24.6250,0.0000
C01299=43.571,40.607,66.599,-153.7793,-25.7759,0.0000
C01300=45.409,38.659,66.632,-153.3982,-25.1992,0.0000
C01301=48.211,36.955,67.386,-151.5860,-21.9235,0.0000
C01302=51.344,38.042,69.285,-150.8323,-19.7582,0.0000
C01303=55.523,41.042,71.901,-150.2510,-17.3162,0.0000
C01304=60.870,45.159,74.567,-150.3196,-11.9799,0.0000
C01305=66.782,49.709,76.575,-172.6970,2.7884,0.0000
C01306=72.396,53.692,77.551,177.6244,-1.4685,0.0000
C01307=78.373,54.731,78.062,175.7429,-2.7669,0.0000
C01308=83.926,52.567,78.476,174.9940,-3.2736,0.0000
C01309=87.904,47.632,78.891,174.8913,-3.3329,0.0000
C01310=90.984,41.489,79.163,175.0845,-3.1947,0.0000
C01311=93.673,34.998,79.163,-174.2652,1.2084,0.0000
C01312=95.839,28.477,78.891,-174.0309,1.2462,0.0000
C01313=96.515,22.174,78.476,-174.1455,1.2161,0.0000
C01314=94.118,16.717,78.062,-175.0332,1.0483,0.0000
C01315=89.158,13.226,77.551,-177.2817,0.6405,0.0000
C01316=82.372,12.073,76.575,172.8558,-3.1745,0.0000
C01317=74.974,11.109,74.567,167.0303,-29.2929,0.0000
C01318=68.282,10.239,71.901,171.4578,-33.0541,0.0000
C01319=63.206,9.406,69.285,174.0746,-34.2892,0.0000
C01320=60.221,7.959,67.386,176.6249,-35.1801,0.0000
C01321=59.445,4.772,66.632,-178.9672,-35.9843,0.0000
C01322=59.523,2.097,66.599,-178.1470,-36.0735,0.0000
C01323=59.554,0.000,66.621,-179.9989,-36.1063,0.0000
C01324=59.523,-2.096,66.599,178.1458,-36.0735,0.0000
C01325=59.445,-4.772,66.632,178.9688,-35.9842,0.0000
C01326=60.222,-7.959,67.386,-176.6244,-35.1800,0.0000
C01327=63.206,-9.406,69.285,-174.0744,-34.2892,0.0000
C01328=68.282,-10.239,71.901,-171.4578,-33.0542,0.0000
C01329=74.974,-11.109,74.567,-167.0305,-29.2932,0.0000
C01330=82.372,-12.073,76.575,-172.8557,-3.1746,0.0000
C01331=89.158,-13.226,77.551,177.2817,0.6405,0.0000
C01332=94.118,-16.717,78.062,175.0332,1.0483,0.0000
C01333=96.515,-22.174,78.476,174.1455,1.2161,0.0000
C01334=95.839,-28.477,78.891,174.0309,1.2462,0.0000
C01335=93.673,-34.998,79.163,174.2652,1.2084,0.0000
C01336=90.984,-41.489,79.163,-175.0845,-3.1947,0.0000
C01337=87.904,-47.632,78.891,-174.8913,-3.3329,0.0000
C01338=83.926,-52.567,78.476,-174.9940,-3.2736,0.0000
C01339=78.373,-54.731,78.062,-175.7429,-2.7669,0.0000
C01340=72.396,-53.692,77.551,-177.6244,-1.4685,0.0000
C01341=66.782,-49.709,76.575,172.6972,2.7884,0.0000
C01342=60.870,-45.159,74.567,150.3197,-11.9795,0.0000
C01343=55.523,-41.042,71.901,150.2510,-17.3162,0.0000
C01344=51.344,-38.042,69.285,150.8323,-19.7583,0.0000
C01345=48.211,-36.955,67.386,151.5862,-21.9238,0.0000
C01346=45.408,-38.660,66.632,153.3991,-25.2003,0.0000
C01347=43.572,-40.607,66.599,153.7787,-25.7752,0.0000
C01348=42.111,-42.111,66.621,152.7181,-24.6263,0.0000
C01349=40.607,-43.571,66.599,151.7068,-23.4450,0.0000
C01350=38.659,-45.409,66.632,152.2441,-23.9019,0.0000
C01351=36.955,-48.211,67.386,155.4112,-26.1950,0.0000
C01352=38.042,-51.344,69.285,157.6397,-27.3017,0.0000
C01353=41.042,-55.523,71.901,160.2466,-28.2755,0.0000
C01354=45.159,-60.870,74.567,166.2752,-28.9717,0.0000
C01355=49.709,-66.782,76.575,-177.1888,-7.2943,0.0000
C01356=53.692,-72.396,77.551,178.5302,2.3748,0.0000
C01357=54.731,-78.373,78.062,177.2254,4.2522,0.0000
C01358=52.567,-83.926,78.476,176.7139,4.9979,0.0000
C01359=47.632,-87.904,78.891,176.6538,5.1000,0.0000
C01360=41.489,-90.984,79.163,176.7935,4.9078,0.0000
C01361=34.998,-93.673,79.163,-178.7855,-5.7335,0.0000
C01362=28.477,-95.839,78.891,-178.7470,-5.9677,0.0000
C01363=22.174,-96.515,78.476,-178.7775,-5.8532,0.0000
C01364=16.717,-94.118,78.062,-178.9478,-4.9659,0.0000
C01365=13.226,-89.158,77.551,-179.3588,-2.7181,0.0000
C01366=12.073,-82.372,76.575,176.8007,7.1331,0.0000
C01367=11.109,-74.974,74.567,150.0710,11.2878,0.0000
C01368=10.239,-68.282,71.901,146.6530,7.1518,0.0000
C01369=9.406,-63.206,69.285,145.5678,4.8928,0.0000
C01370=7.959,-60.221,67.386,144.7730,2.7581,0.0000
C01371=4.772,-59.445,66.632,144.0113,-0.8357,0.0000
C01372=2.097,-59.523,66.599,143.9122,-1.4976,0.0000
C01373=0.000,-59.554,66.621,143.8937,-0.0009,0.0000
C01374=0.000,-59.554,66.621,143.8937,-0.0009,0.0000
C01375=-2.096,-59.523,66.599,143.9122,1.4986,0.0000
C01376=-4.772,-59.445,66.632,144.0114,0.8344,0.0000
C01377=-7.959,-60.222,67.386,144.7731,-2.7585,0.0000
C01378=-9.406,-63.206,69.285,145.5678,-4.8929,0.0000
C01379=-10.239,-68.282,71.901,146.6530,-7.1518,0.0000
C01380=-11.109,-74.974,74.567,150.0708,-11.2876,0.0000
C01381=-12.073,-82.372,76.575,176.8006,-7.1333,0.0000
C01382=-13.226,-89.158,77.551,-179.3588,2.7181,0.0000
C01383=-16.717,-94.118,78.062,-178.9478,4.9659,0.0000
C01384=-22.174,-96.515,78.476,-178.7775,5.8532,0.0000
C01385=-28.477,-95.839,78.891,-178.7470,5.9677,0.0000
C01386=-34.998,-93.673,79.163,-178.7855,5.7335,0.0000
C01387=-41.489,-90.984,79.163,176.7935,-4.9078,0.0000
C01388=-47.632,-87.904,78.891,176.6538,-5.1000,0.0000
C01389=-52.567,-83.926,78.476,176.7139,-4.9979,0.0000
C01390=-54.731,-78.373,78.062,177.2254,-4.2522,0.0000
C01391=-53.692,-72.396,77.551,178.5302,-2.3748,0.0000
C01392=-49.709,-66.782,76.575,-177.1888,7.2941,0.0000
C01393=-45.159,-60.870,74.567,166.2756,28.9717,0.0000
C01394=-41.042,-55.523,71.901,160.2467,28.2755,0.0000
C01395=-38.042,-51.344,69.285,157.6396,27.3016,0.0000
C01396=-36.955,-48.211,67.386,155.4109,26.1948,0.0000
C01397=-38.660,-45.408,66.632,152.2432,23.9010,0.0000
C01398=-40.607,-43.572,66.599,151.7075,23.4457,0.0000
C01399=-42.111,-42.111,66.621,152.7169,24.6250,0.0000
C01400=-43.571,-40.607,66.599,153.7793,25.7759,0.0000
C01401=-45.409,-38.659,66.632,153.3982,25.1992,0.0000
C01402=-48.211,-36.955,67.386,151.5860,21.9235,0.0000
C01403=-51.344,-38.042,69.285,150.8323,19.7582,0.0000
C01404=-55.523,-41.042,71.901,150.2510,17.3162,0.0000
C01405=-60.870,-45.159,74.567,150.3196,11.9799,0.0000
C01406=-66.782,-49.709,76.575,172.6970,-2.7884,0.0000
C01407=-72.396,-53.692,77.551,-177.6244,1.4685,0.0000
C01408=-78.373,-54.731,78.062,-175.7429,2.7669,0.0000
C01409=-83.926,-52.567,78.476,-174.9940,3.2736,0.0000
C01410=-87.904,-47.632,78.891,-174.8913,3.3329,0.0000
C01411=-90.984,-41.489,79.163,-175.0845,3.1947,0.0000
C01412=-93.673,-34.998,79.163,174.2652,-1.2084,0.0000
C01413=-95.839,-28.477,78.891,174.0309,-1.2462,0.0000
C01414=-96.515,-22.174,78.476,174.1455,-1.2161,0.0000
C01415=-94.118,-16.717,78.062,175.0332,-1.0483,0.0000
C01416=-89.158,-13.226,77.551,177.2817,-0.6405,0.0000
C01417=-82.372,-12.073,76.575,-172.8558,3.1745,0.0000
C01418=-74.974,-11.109,74.567,-167.0303,29.2929,0.0000
C01419=-68.282,-10.239,71.901,-171.4578,33.0541,0.0000
C01420=-63.206,-9.406,69.285,-174.0746,34.2892,0.0000
C01421=-60.221,-7.959,67.386,-176.6249,35.1801,0.0000
C01422=-59.445,-4.772,66.632,178.9672,35.9843,0.0000
C01423=-59.523,-2.097,66.599,178.1470,36.0735,0.0000
C01424=-59.554,0.000,66.621,179.9989,36.1063,0.0000
C01425=-59.523,2.096,66.599,-178.1458,36.0735,0.0000
C01426=-59.445,4.772,66.632,-178.9688,35.9842,0.0000
C01427=-60.222,7.959,67.386,176.6244,35.1800,0.0000
C01428=-63.206,9.406,69.285,174.0744,34.2892,0.0000
C01429=-68.282,10.239,71.901,171.4578,33.0542,0.0000
C01430=-74.974,11.109,74.567,167.0305,29.2932,0.0000
C01431=-82.372,12.073,76.575,172.8557,3.1746,0.0000
C01432=-89.158,13.226,77.551,-177.2817,-0.6405,0.0000
C01433=-94.118,16.717,78.062,-175.0332,-1.0483,0.0000
C01434=-96.515,22.174,78.476,-174.1455,-1.2161,0.0000
C01435=-95.839,28.477,78.891,-174.0309,-1.2462,0.0000
C01436=-93.673,34.998,79.163,-174.2652,-1.2084,0.0000
C01437=-90.984,41.489,79.163,175.0845,3.1947,0.0000
C01438=-87.904,47.632,78.891,174.8913,3.3329,0.0000
C01439=-83.926,52.567,78.476,174.9940,3.2736,0.0000
C01440=-78.373,54.731,78.062,175.7429,2.7669,0.0000
C01441=-72.396,53.692,77.551,177.6244,1.4685,0.0000
C01442=-66.782,49.709,76.575,-172.6972,-2.7884,0.0000
C01443=-60.870,45.159,74.567,-150.3197,11.9795,0.0000
C01444=-55.523,41.042,71.901,-150.2510,17.3162,0.0000
C01445=-51.344,38.042,69.285,-150.8323,19.7583,0.0000
C01446=-48.211,36.955,67.386,-151.5862,21.9238,0.0000
C01447=-45.408,38.660,66.632,-153.3991,25.2003,0.0000
C01448=-43.572,40.607,66.599,-153.7787,25.7752,0.0000
C01449=-42.111,42.111,66.621,-152.7181,24.6263,0.0000
C01450=-40.607,43.571,66.599,-151.7068,23.4450,0.0000
C01451=-38.659,45.409,66.632,-152.2441,23.9019,0.0000
C01452=-36.955,48.211,67.386,-155.4112,26.1950,0.0000
C01453=-38.042,51.344,69.285,-157.6397,27.3017,0.0000
C01454=-41.042,55.523,71.901,-160.2466,28.2755,0.0000
C01455=-45.159,60.870,74.567,-166.2752,28.9717,0.0000
C01456=-49.709,66.782,76.575,177.1888,7.2943,0.0000
C01457=-53.692,72.396,77.551,-178.5302,-2.3748,0.0000
C01458=-54.731,78.373,78.062,-177.2254,-4.2522,0.0000
C01459=-52.567,83.926,78.476,-176.7139,-4.9979,0.0000
C01460=-47.632,87.904,78.891,-176.6538,-5.1000,0.0000
C01461=-41.489,90.984,79.163,-176.7935,-4.9078,0.0000
C01462=-34.998,93.673,79.163,178.7855,5.7335,0.0000
C01463=-28.477,95.839,78.891,178.7470,5.9677,0.0000
C01464=-22.174,96.515,78.476,178.7775,5.8532,0.0000
C01465=-16.717,94.118,78.062,178.9478,4.9659,0.0000
C01466=-13.226,89.158,77.551,179.3588,2.7181,0.0000
C01467=-12.073,82.372,76.575,-176.8006,-7.1333,0.0000
C01468=-11.109,74.974,74.567,-150.0708,-11.2876,0.0000
C01469=-10.239,68.282,71.901,-146.6530,-7.1518,0.0000
C01470=-9.406,63.206,69.285,-145.5678,-4.8929,0.0000
C01471=-7.959,60.222,67.386,-144.7731,-2.7585,0.0000
C01472=-4.772,59.445,66.632,-144.0114,0.8344,0.0000
C01473=-2.096,59.523,66.599,-143.9122,1.4986,0.0000
C01474=0.000,59.554,66.621,-143.8937,-0.0009,0.0000
C01475=0.000,58.319,68.442,-144.4660,-0.0009,0.0000
C01476=1.984,58.291,68.419,-144.4831,-1.4398,0.0000
C01477=4.582,58.225,68.453,-144.5791,-0.8115,0.0000
C01478=7.730,59.058,69.238,-145.3357,2.7529,0.0000
C01479=9.135,62.185,71.215,-146.1245,4.8662,0.0000
C01480=9.949,67.473,73.927,-147.2558,7.2044,0.0000
C01481=10.820,74.409,76.674,-151.2143,11.6876,0.0000
C01482=11.787,82.032,78.729,-179.1416,2.6765,0.0000
C01483=12.929,88.996,79.725,179.2461,-3.4524,0.0000
C01484=16.445,94.085,80.245,178.9321,-5.3082,0.0000
C01485=21.964,96.553,80.665,178.7840,-6.0851,0.0000
C01486=28.347,95.882,81.086,178.7564,-6.1844,0.0000
C01487=34.955,93.690,81.363,178.7907,-5.9678,0.0000
C01488=41.532,90.965,81.363,-176.6230,5.0693,0.0000
C01489=47.755,87.843,81.086,-176.4928,5.2460,0.0000
C01490=52.743,83.804,80.665,-176.5441,5.1566,0.0000
C01491=54.900,78.157,80.245,-176.9931,4.5046,0.0000
C01492=53.787,72.072,79.725,-178.0895,2.9732,0.0000
C01493=49.670,66.340,78.729,178.7131,-2.4989,0.0000
C01494=44.964,60.266,76.674,-167.5049,-28.4687,0.0000
C01495=40.676,54.746,73.927,-160.7888,-27.9126,0.0000
C01496=37.512,50.430,71.215,-158.0896,-26.9169,0.0000
C01497=36.294,47.226,69.238,-155.8851,-25.8283,0.0000
C01498=37.931,44.411,68.453,-152.7428,-23.5637,0.0000
C01499=39.816,42.621,68.419,-152.2321,-23.1346,0.0000
C01500=41.238,41.238,68.442,-153.2052,-24.2645,0.0000
C01501=42.621,39.816,68.419,-154.2270,-25.3685,0.0000
C01502=44.412,37.931,68.453,-153.8660,-24.8207,0.0000
C01503=47.226,36.294,69.238,-152.0624,-21.5768,0.0000
C01504=50.430,37.512,71.215,-151.3113,-19.4345,0.0000
C01505=54.746,40.676,73.927,-150.7077,-16.9041,0.0000
C01506=60.266,44.964,76.674,-150.9519,-10.9645,0.0000
C01507=66.340,49.670,78.729,-177.5004,1.2857,0.0000
C01508=72.072,53.787,79.725,177.0252,-1.9079,0.0000
C01509=78.157,54.900,80.245,175.4892,-2.9976,0.0000
C01510=83.804,52.743,80.665,174.8340,-3.4419,0.0000
C01511=87.843,47.755,81.086,174.7442,-3.4925,0.0000
C01512=90.965,41.532,81.363,174.9219,-3.3638,0.0000
C01513=93.690,34.955,81.363,-174.0309,1.2028,0.0000
C01514=95.882,28.347,81.086,-173.8142,1.2363,0.0000
C01515=96.553,21.964,80.665,-173.9135,1.2091,0.0000
C01516=94.085,16.445,80.245,-174.6909,1.0633,0.0000
C01517=88.996,12.929,79.725,-176.5473,0.7526,0.0000
C01518=82.032,11.787,78.729,177.3232,-0.8574,0.0000
C01519=74.409,10.820,76.674,166.7195,-28.1350,0.0000
C01520=67.473,9.949,73.927,171.4531,-32.4538,0.0000
C01521=62.185,9.135,71.215,174.1452,-33.7370,0.0000
C01522=59.058,7.730,69.238,176.6542,-34.6185,0.0000
C01523=58.225,4.582,68.453,-179.0043,-35.4168,0.0000
C01524=58.291,1.984,68.419,-178.2313,-35.5040,0.0000
C01525=58.319,0.000,68.442,-179.9988,-35.5340,0.0000
C01526=58.291,-1.983,68.419,178.2301,-35.5040,0.0000
C01527=58.225,-4.583,68.453,179.0058,-35.4167,0.0000
C01528=59.058,-7.730,69.238,-176.6538,-34.6185,0.0000
C01529=62.185,-9.135,71.215,-174.1451,-33.7370,0.0000
C01530=67.473,-9.949,73.927,-171.4531,-32.4539,0.0000
C01531=74.409,-10.820,76.674,-166.7196,-28.1353,0.0000
C01532=82.032,-11.787,78.729,-177.3232,-0.8574,0.0000
C01533=88.996,-12.929,79.725,176.5473,0.7526,0.0000
C01534=94.085,-16.445,80.245,174.6909,1.0633,0.0000
C01535=96.553,-21.964,80.665,173.9135,1.2091,0.0000
C01536=95.882,-28.347,81.086,173.8142,1.2363,0.0000
C01537=93.690,-34.955,81.363,174.0309,1.2028,0.0000
C01538=90.965,-41.532,81.363,-174.9219,-3.3638,0.0000
C01539=87.843,-47.755,81.086,-174.7442,-3.4925,0.0000
C01540=83.804,-52.743,80.665,-174.8340,-3.4419,0.0000
C01541=78.157,-54.900,80.245,-175.4892,-2.9976,0.0000
C01542=72.072,-53.787,79.725,-177.0252,-1.9079,0.0000
C01543=66.340,-49.670,78.729,177.5004,1.2857,0.0000
C01544=60.266,-44.964,76.674,150.9520,-10.9641,0.0000
C01545=54.746,-40.676,73.927,150.7078,-16.9040,0.0000
C01546=50.430,-37.512,71.215,151.3114,-19.4346,0.0000
C01547=47.226,-36.294,69.238,152.0626,-21.5771,0.0000
C01548=44.411,-37.931,68.453,153.8669,-24.8217,0.0000
C01549=42.621,-39.816,68.419,154.2263,-25.3677,0.0000
C01550=41.238,-41.238,68.442,153.2065,-24.2659,0.0000
C01551=39.816,-42.621,68.419,152.2314,-23.1338,0.0000
C01552=37.931,-44.412,68.453,152.7438,-23.5646,0.0000
C01553=36.294,-47.226,69.238,155.8855,-25.8286,0.0000
C01554=37.512,-50.430,71.215,158.0896,-26.9170,0.0000
C01555=40.676,-54.746,73.927,160.7888,-27.9127,0.0000
C01556=44.964,-60.266,76.674,167.5045,-28.4688,0.0000
C01557=49.670,-66.340,78.729,-178.7131,-2.4989,0.0000
C01558=53.787,-72.072,79.725,178.0895,2.9732,0.0000
C01559=54.900,-78.157,80.245,176.9931,4.5046,0.0000
C01560=52.743,-83.804,80.665,176.5441,5.1566,0.0000
C01561=47.755,-87.843,81.086,176.4928,5.2460,0.0000
C01562=41.532,-90.965,81.363,176.6230,5.0693,0.0000
C01563=34.955,-93.690,81.363,-178.7907,-5.9678,0.0000
C01564=28.347,-95.882,81.086,-178.7564,-6.1844,0.0000
C01565=21.964,-96.553,80.665,-178.7840,-6.0851,0.0000
C01566=16.445,-94.085,80.245,-178.9321,-5.3082,0.0000
C01567=12.929,-88.996,79.725,-179.2461,-3.4524,0.0000
C01568=11.787,-82.032,78.729,179.1416,2.6765,0.0000
C01569=10.820,-74.409,76.674,151.2143,11.6876,0.0000
C01570=9.949,-67.473,73.927,147.2558,7.2044,0.0000
C01571=9.135,-62.185,71.215,146.1245,4.8662,0.0000
C01572=7.730,-59.058,69.238,145.3357,2.7529,0.0000
C01573=4.582,-58.225,68.453,144.5791,-0.8115,0.0000
C01574=1.984,-58.291,68.419,144.4831,-1.4398,0.0000
C01575=0.000,-58.319,68.442,144.4660,-0.0009,0.0000
C01576=0.000,-58.319,68.442,144.4660,-0.0009,0.0000
C01577=-1.983,-58.291,68.419,144.4831,1.4408,0.0000
C01578=-4.583,-58.225,68.453,144.5792,0.8102,0.0000
C01579=-7.730,-59.058,69.238,145.3358,-2.7533,0.0000
C01580=-9.135,-62.185,71.215,146.1245,-4.8663,0.0000
C01581=-9.949,-67.473,73.927,147.2557,-7.2044,0.0000
C01582=-10.820,-74.409,76.674,151.2140,-11.6874,0.0000
C01583=-11.787,-82.032,78.729,179.1416,-2.6765,0.0000
C01584=-12.929,-88.996,79.725,-179.2461,3.4524,0.0000
C01585=-16.445,-94.085,80.245,-178.9321,5.3082,0.0000
C01586=-21.964,-96.553,80.665,-178.7840,6.0851,0.0000
C01587=-28.347,-95.882,81.086,-178.7564,6.1844,0.0000
C01588=-34.955,-93.690,81.363,-178.7907,5.9678,0.0000
C01589=-41.532,-90.965,81.363,176.6230,-5.0693,0.0000
C01590=-47.755,-87.843,81.086,176.4928,-5.2460,0.0000
C01591=-52.743,-83.804,80.665,176.5441,-5.1566,0.0000
C01592=-54.900,-78.157,80.245,176.9931,-4.5046,0.0000
C01593=-53.787,-72.072,79.725,178.0895,-2.9732,0.0000
C01594=-49.670,-66.340,78.729,-178.7131,2.4989,0.0000
C01595=-44.964,-60.266,76.674,167.5049,28.4687,0.0000
C01596=-40.676,-54.746,73.927,160.7888,27.9126,0.0000
C01597=-37.512,-50.430,71.215,158.0896,26.9169,0.0000
C01598=-36.294,-47.226,69.238,155.8851,25.8283,0.0000
C01599=-37.931,-44.411,68.453,152.7428,23.5637,0.0000
C01600=-39.816,-42.621,68.419,152.2321,23.1346,0.0000
C01601=-41.238,-41.238,68.442,153.2052,24.2645,0.0000
C01602=-42.621,-39.816,68.419,154.2270,25.3685,0.0000
C01603=-44.412,-37.931,68.453,153.8660,24.8207,0.0000
C01604=-47.226,-36.294,69.238,152.0624,21.5768,0.0000
C01605=-50.430,-37.512,71.215,151.3113,19.4345,0.0000
C01606=-54.746,-40.676,73.927,150.7077,16.9041,0.0000
C01607=-60.266,-44.964,76.674,150.9519,10.9645,0.0000
C01608=-66.340,-49.670,78.729,177.5004,-1.2857,0.0000
C01609=-72.072,-53.787,79.725,-177.0252,1.9079,0.0000
C01610=-78.157,-54.900,80.245,-175.4892,2.9976,0.0000
C01611=-83.804,-52.743,80.665,-174.8340,3.4419,0.0000
C01612=-87.843,-47.755,81.086,-174.7442,3.4925,0.0000
C01613=-90.965,-41.532,81.363,-174.9219,3.3638,0.0000
C01614=-93.690,-34.955,81.363,174.0309,-1.2028,0.0000
C01615=-95.882,-28.347,81.086,173.8142,-1.2363,0.0000
C01616=-96.553,-21.964,80.665,173.9135,-1.2091,0.0000
C01617=-94.085,-16.445,80.245,174.6909,-1.0633,0.0000
C01618=-88.996,-12.929,79.725,176.5473,-0.7526,0.0000
C01619=-82.032,-11.787,78.729,-177.3232,0.8574,0.0000
C01620=-74.409,-10.820,76.674,-166.7195,28.1350,0.0000
C01621=-67.473,-9.949,73.927,-171.4531,32.4538,0.0000
C01622=-62.185,-9.135,71.215,-174.1452,33.7370,0.0000
C01623=-59.058,-7.730,69.238,-176.6542,34.6185,0.0000
C01624=-58.225,-4.582,68.453,179.0043,35.4168,0.0000
C01625=-58.291,-1.984,68.419,178.2313,35.5040,0.0000
C01626=-58.319,0.000,68.442,179.9988,35.5340,0.0000
C01627=-58.291,1.983,68.419,-178.2301,35.5040,0.0000
C01628=-58.225,4.583,68.453,-179.0058,35.4167,0.0000
C01629=-59.058,7.730,69.238,176.6538,34.6185,0.0000
C01630=-62.185,9.135,71.215,174.1451,33.7370,0.0000
C01631=-67.473,9.949,73.927,171.4531,32.4539,0.0000
C01632=-74.409,10.820,76.674,166.7196,28.1353,0.0000
C01633=-82.032,11.787,78.729,177.3232,0.8574,0.0000
C01634=-88.996,12.929,79.725,-176.5473,-0.7526,0.0000
C01635=-94.085,16.445,80.245,-174.6909,-1.0633,0.0000
C01636=-96.553,21.964,80.665,-173.9135,-1.2091,0.0000
C01637=-95.882,28.347,81.086,-173.8142,-1.2363,0.0000
C01638=-93.690,34.955,81.363,-174.0309,-1.2028,0.0000
C01639=-90.965,41.532,81.363,174.9219,3.3638,0.0000
C01640=-87.843,47.755,81.086,174.7442,3.4925,0.0000
C01641=-83.804,52.743,80.665,174.8340,3.4419,0.0000
C01642=-78.157,54.900,80.245,175.4892,2.9976,0.0000
C01643=-72.072,53.787,79.725,177.0252,1.9079,0.0000
C01644=-66.340,49.670,78.729,-177.5004,-1.2857,0.0000
C01645=-60.266,44.964,76.674,-150.9520,10.9641,0.0000
C01646=-54.746,40.676,73.927,-150.7078,16.9040,0.0000
C01647=-50.430,37.512,71.215,-151.3114,19.4346,0.0000
C01648=-47.226,36.294,69.238,-152.0626,21.5771,0.0000
C01649=-44.411,37.931,68.453,-153.8669,24.8217,0.0000
C01650=-42.621,39.816,68.419,-154.2263,25.3677,0.0000
C01651=-41.238,41.238,68.442,-153.2065,24.2659,0.0000
C01652=-39.816,42.621,68.419,-152.2314,23.1338,0.0000
C01653=-37.931,44.412,68.453,-152.7438,23.5646,0.0000
C01654=-36.294,47.226,69.238,-155.8855,25.8286,0.0000
C01655=-37.512,50.430,71.215,-158.0896,26.9170,0.0000
C01656=-40.676,54.746,73.927,-160.7888,27.9127,0.0000
C01657=-44.964,60.266,76.674,-167.5045,28.4688,0.0000
C01658=-49.670,66.340,78.729,178.7131,2.4989,0.0000
C01659=-53.787,72.072,79.725,-178.0895,-2.9732,0.0000
C01660=-54.900,78.157,80.245,-176.9931,-4.5046,0.0000
C01661=-52.743,83.804,80.665,-176.5441,-5.1566,0.0000
C01662=-47.755,87.843,81.086,-176.4928,-5.2460,0.0000
C01663=-41.532,90.965,81.363,-176.6230,-5.0693,0.0000
C01664=-34.955,93.690,81.363,178.7907,5.9678,0.0000
C01665=-28.347,95.882,81.086,178.7564,6.1844,0.0000
C01666=-21.964,96.553,80.665,178.7840,6.0851,0.0000
C01667=-16.445,94.085,80.245,178.9321,5.3082,0.0000
C01668=-12.929,88.996,79.725,179.2461,3.4524,0.0000
C01669=-11.787,82.032,78.729,-179.1416,-2.6765,0.0000
C01670=-10.820,74.409,76.674,-151.2140,-11.6874,0.0000
C01671=-9.949,67.473,73.927,-147.2557,-7.2044,0.0000
C01672=-9.135,62.185,71.215,-146.1245,-4.8663,0.0000
C01673=-7.730,59.058,69.238,-145.3358,-2.7533,0.0000
C01674=-4.583,58.225,68.453,-144.5792,0.8102,0.0000
C01675=-1.983,58.291,68.419,-144.4831,1.4408,0.0000
C01676=0.000,58.319,68.442,-144.4660,-0.0009,0.0000
C01677=0.000,57.118,70.285,-145.0906,-0.0010,0.0000
C01678=1.874,57.094,70.261,-145.1062,-1.3791,0.0000
C01679=4.398,57.039,70.297,-145.1991,-0.7888,0.0000
C01680=7.507,57.930,71.114,-145.9507,2.7407,0.0000
C01681=8.875,61.204,73.167,-146.7377,4.8362,0.0000
C01682=9.674,66.709,75.971,-147.9316,7.2677,0.0000
C01683=10.553,73.885,78.794,-152.6143,12.1344,0.0000
C01684=11.527,81.722,80.892,-179.8231,0.6439,0.0000
C01685=12.662,88.851,81.904,179.1858,-3.9847,0.0000
C01686=16.202,94.056,82.431,178.9359,-5.5425,0.0000
C01687=21.776,96.587,82.857,178.8046,-6.2332,0.0000
C01688=28.231,95.920,83.283,178.7790,-6.3232,0.0000
C01689=34.916,93.705,83.562,178.8092,-6.1263,0.0000
C01690=41.570,90.949,83.562,-176.4970,5.1678,0.0000
C01691=47.863,87.788,83.283,-176.3779,5.3278,0.0000
C01692=52.900,83.695,82.857,-176.4241,5.2464,0.0000
C01693=55.051,77.964,82.431,-176.8237,4.6670,0.0000
C01694=53.873,71.781,81.904,-177.7544,3.3917,0.0000
C01695=49.635,65.937,80.892,179.6697,-0.5804,0.0000
C01696=44.783,59.707,78.794,-168.9613,-27.8155,0.0000
C01697=40.330,54.011,75.971,-161.3963,-27.5073,0.0000
C01698=37.003,49.553,73.167,-158.5816,-26.4913,0.0000
C01699=35.654,46.271,71.114,-156.3955,-25.4213,0.0000
C01700=37.223,43.442,70.297,-153.2828,-23.1907,0.0000
C01701=39.047,41.697,70.261,-152.8002,-22.7910,0.0000
C01702=40.388,40.388,70.285,-153.7349,-23.8693,0.0000
C01703=41.696,39.047,70.261,-154.7139,-24.9243,0.0000
C01704=43.443,37.223,70.297,-154.3761,-24.4088,0.0000
C01705=46.271,35.654,71.114,-152.5845,-21.2012,0.0000
C01706=49.553,37.003,73.167,-151.8368,-19.0766,0.0000
C01707=54.011,40.330,75.971,-151.2139,-16.4368,0.0000
C01708=59.707,44.783,78.794,-151.7405,-9.7503,0.0000
C01709=65.937,49.635,80.892,-179.4196,0.3303,0.0000
C01710=71.781,53.873,81.904,176.6057,-2.2416,0.0000
C01711=77.964,55.051,82.431,175.3258,-3.1657,0.0000
C01712=83.695,52.900,82.857,174.7434,-3.5609,0.0000
C01713=87.788,47.863,83.283,174.6616,-3.6065,0.0000
C01714=90.949,41.570,83.562,174.8225,-3.4887,0.0000
C01715=93.705,34.916,83.562,-173.8724,1.1840,0.0000
C01716=95.920,28.231,83.283,-173.6754,1.2135,0.0000
C01717=96.587,21.776,82.857,-173.7655,1.1884,0.0000
C01718=94.056,16.202,82.431,-174.4566,1.0591,0.0000
C01719=88.851,12.662,81.904,-176.0149,0.8122,0.0000
C01720=81.722,11.527,80.892,179.3561,-0.1768,0.0000
C01721=73.885,10.553,78.794,166.3880,-26.7245,0.0000
C01722=66.709,9.674,75.971,171.4416,-31.7804,0.0000
C01723=61.204,8.875,73.167,174.2221,-33.1286,0.0000
C01724=57.930,7.507,71.114,176.6934,-34.0050,0.0000
C01725=57.039,4.398,70.297,-179.0395,-34.7972,0.0000
C01726=57.094,1.874,70.261,-178.3187,-34.8823,0.0000
C01727=57.118,0.000,70.285,-179.9988,-34.9094,0.0000
C01728=57.094,-1.874,70.261,178.3174,-34.8823,0.0000
C01729=57.039,-4.398,70.297,179.0410,-34.7971,0.0000
C01730=57.930,-7.507,71.114,-176.6929,-34.0050,0.0000
C01731=61.204,-8.875,73.167,-174.2220,-33.1286,0.0000
C01732=66.709,-9.674,75.971,-171.4416,-31.7805,0.0000
C01733=73.885,-10.553,78.794,-166.3881,-26.7249,0.0000
C01734=81.722,-11.527,80.892,-179.3561,-0.1768,0.0000
C01735=88.851,-12.662,81.904,176.0149,0.8122,0.0000
C01736=94.056,-16.202,82.431,174.4566,1.0591,0.0000
C01737=96.587,-21.776,82.857,173.7655,1.1884,0.0000
C01738=95.920,-28.231,83.283,173.6754,1.2135,0.0000
C01739=93.705,-34.916,83.562,173.8724,1.1840,0.0000
C01740=90.949,-41.570,83.562,-174.8225,-3.4887,0.0000
C01741=87.788,-47.863,83.283,-174.6616,-3.6065,0.0000
C01742=83.695,-52.900,82.857,-174.7434,-3.5609,0.0000
C01743=77.964,-55.051,82.431,-175.3258,-3.1657,0.0000
C01744=71.781,-53.873,81.904,-176.6057,-2.2416,0.0000
C01745=65.937,-49.635,80.892,179.4196,0.3303,0.0000
C01746=59.707,-44.783,78.794,151.7406,-9.7500,0.0000
C01747=54.011,-40.330,75.971,151.2139,-16.4367,0.0000
C01748=49.553,-37.003,73.167,151.8369,-19.0767,0.0000
C01749=46.271,-35.654,71.114,152.5847,-21.2016,0.0000
C01750=43.442,-37.223,70.297,154.3770,-24.4098,0.0000
C01751=41.697,-39.047,70.261,154.7132,-24.9235,0.0000
C01752=40.388,-40.388,70.285,153.7363,-23.8708,0.0000
C01753=39.047,-41.696,70.261,152.7994,-22.7901,0.0000
C01754=37.223,-43.443,70.297,153.2837,-23.1916,0.0000
C01755=35.654,-46.271,71.114,156.3959,-25.4216,0.0000
C01756=37.003,-49.553,73.167,158.5816,-26.4914,0.0000
C01757=40.330,-54.011,75.971,161.3962,-27.5073,0.0000
C01758=44.783,-59.707,78.794,168.9608,-27.8156,0.0000
C01759=49.635,-65.937,80.892,-179.6697,-0.5804,0.0000
C01760=53.873,-71.781,81.904,177.7544,3.3917,0.0000
C01761=55.051,-77.964,82.431,176.8237,4.6670,0.0000
C01762=52.900,-83.695,82.857,176.4241,5.2464,0.0000
C01763=47.863,-87.788,83.283,176.3779,5.3278,0.0000
C01764=41.570,-90.949,83.562,176.4970,5.1678,0.0000
C01765=34.916,-93.705,83.562,-178.8092,-6.1263,0.0000
C01766=28.231,-95.920,83.283,-178.7790,-6.3232,0.0000
C01767=21.776,-96.587,82.857,-178.8046,-6.2332,0.0000
C01768=16.202,-94.056,82.431,-178.9359,-5.5425,0.0000
C01769=12.662,-88.851,81.904,-179.1858,-3.9847,0.0000
C01770=11.527,-81.722,80.892,179.8231,0.6439,0.0000
C01771=10.553,-73.885,78.794,152.6143,12.1344,0.0000
C01772=9.674,-66.709,75.971,147.9316,7.2677,0.0000
C01773=8.875,-61.204,73.167,146.7377,4.8362,0.0000
C01774=7.507,-57.930,71.114,145.9507,2.7407,0.0000
C01775=4.398,-57.039,70.297,145.1991,-0.7888,0.0000
C01776=1.874,-57.094,70.261,145.1062,-1.3791,0.0000
C01777=0.000,-57.118,70.285,145.0906,-0.0010,0.0000
C01778=0.000,-57.118,70.285,145.0906,-0.0010,0.0000
C01779=-1.874,-57.094,70.261,145.1061,1.3802,0.0000
C01780=-4.398,-57.039,70.297,145.1991,0.7875,0.0000
C01781=-7.507,-57.930,71.114,145.9507,-2.7411,0.0000
C01782=-8.875,-61.204,73.167,146.7377,-4.8363,0.0000
C01783=-9.674,-66.709,75.971,147.9315,-7.2677,0.0000
C01784=-10.553,-73.885,78.794,152.6139,-12.1342,0.0000
C01785=-11.527,-81.722,80.892,179.8231,-0.6439,0.0000
C01786=-12.662,-88.851,81.904,-179.1858,3.9847,0.0000
C01787=-16.202,-94.056,82.431,-178.9359,5.5425,0.0000
C01788=-21.776,-96.587,82.857,-178.8046,6.2332,0.0000
C01789=-28.231,-95.920,83.283,-178.7790,6.3232,0.0000
C01790=-34.916,-93.705,83.562,-178.8092,6.1263,0.0000
C01791=-41.570,-90.949,83.562,176.4970,-5.1678,0.0000
C01792=-47.863,-87.788,83.283,176.3779,-5.3278,0.0000
C01793=-52.900,-83.695,82.857,176.4241,-5.2464,0.0000
C01794=-55.051,-77.964,82.431,176.8237,-4.6670,0.0000
C01795=-53.873,-71.781,81.904,177.7544,-3.3917,0.0000
C01796=-49.635,-65.937,80.892,-179.6697,0.5804,0.0000
C01797=-44.783,-59.707,78.794,168.9613,27.8155,0.0000
C01798=-40.330,-54.011,75.971,161.3963,27.5073,0.0000
C01799=-37.003,-49.553,73.167,158.5816,26.4913,0.0000
C01800=-35.654,-46.271,71.114,156.3955,25.4213,0.0000
C01801=-37.223,-43.442,70.297,153.2828,23.1907,0.0000
C01802=-39.047,-41.697,70.261,152.8002,22.7910,0.0000
C01803=-40.388,-40.388,70.285,153.7349,23.8693,0.0000
C01804=-41.696,-39.047,70.261,154.7139,24.9243,0.0000
C01805=-43.443,-37.223,70.297,154.3761,24.4088,0.0000
C01806=-46.271,-35.654,71.114,152.5845,21.2012,0.0000
C01807=-49.553,-37.003,73.167,151.8368,19.0766,0.0000
C01808=-54.011,-40.330,75.971,151.2139,16.4368,0.0000
C01809=-59.707,-44.783,78.794,151.7405,9.7503,0.0000
C01810=-65.937,-49.635,80.892,179.4196,-0.3303,0.0000
C01811=-71.781,-53.873,81.904,-176.6057,2.2416,0.0000
C01812=-77.964,-55.051,82.431,-175.3258,3.1657,0.0000
C01813=-83.695,-52.900,82.857,-174.7434,3.5609,0.0000
C01814=-87.788,-47.863,83.283,-174.6616,3.6065,0.0000
C01815=-90.949,-41.570,83.562,-174.8225,3.4887,0.0000
C01816=-93.705,-34.916,83.562,173.8724,-1.1840,0.0000
C01817=-95.920,-28.231,83.283,173.6754,-1.2135,0.0000
C01818=-96.587,-21.776,82.857,173.7655,-1.1884,0.0000
C01819=-94.056,-16.202,82.431,174.4566,-1.0591,0.0000
C01820=-88.851,-12.662,81.904,176.0149,-0.8122,0.0000
C01821=-81.722,-11.527,80.892,-179.3561,0.1768,0.0000
C01822=-73.885,-10.553,78.794,-166.3880,26.7245,0.0000
C01823=-66.709,-9.674,75.971,-171.4416,31.7804,0.0000
C01824=-61.204,-8.875,73.167,-174.2221,33.1286,0.0000
C01825=-57.930,-7.507,71.114,-176.6934,34.0050,0.0000
C01826=-57.039,-4.398,70.297,179.0395,34.7972,0.0000
C01827=-57.094,-1.874,70.261,178.3187,34.8823,0.0000
C01828=-57.118,0.000,70.285,179.9988,34.9094,0.0000
C01829=-57.094,1.874,70.261,-178.3174,34.8823,0.0000
C01830=-57.039,4.398,70.297,-179.0410,34.7971,0.0000
C01831=-57.930,7.507,71.114,176.6929,34.0050,0.0000
C01832=-61.204,8.875,73.167,174.2220,33.1286,0.0000
C01833=-66.709,9.674,75.971,171.4416,31.7805,0.0000
C01834=-73.885,10.553,78.794,166.3881,26.7249,0.0000
C01835=-81.722,11.527,80.892,179.3561,0.1768,0.0000
C01836=-88.851,12.662,81.904,-176.0149,-0.8122,0.0000
C01837=-94.056,16.202,82.431,-174.4566,-1.0591,0.0000
C01838=-96.587,21.776,82.857,-173.7655,-1.1884,0.0000
C01839=-95.920,28.231,83.283,-173.6754,-1.2135,0.0000
C01840=-93.705,34.916,83.562,-173.8724,-1.1840,0.0000
C01841=-90.949,41.570,83.562,174.8225,3.4887,0.0000
C01842=-87.788,47.863,83.283,174.6616,3.6065,0.0000
C01843=-83.695,52.900,82.857,174.7434,3.5609,0.0000
C01844=-77.964,55.051,82.431,175.3258,3.1657,0.0000
C01845=-71.781,53.873,81.904,176.6057,2.2416,0.0000
C01846=-65.937,49.635,80.892,-179.4196,-0.3303,0.0000
C01847=-59.707,44.783,78.794,-151.7406,9.7500,0.0000
C01848=-54.011,40.330,75.971,-151.2139,16.4367,0.0000
C01849=-49.553,37.003,73.167,-151.8369,19.0767,0.0000
C01850=-46.271,35.654,71.114,-152.5847,21.2016,0.0000
C01851=-43.442,37.223,70.297,-154.3770,24.4098,0.0000
C01852=-41.697,39.047,70.261,-154.7132,24.9235,0.0000
C01853=-40.388,40.388,70.285,-153.7363,23.8708,0.0000
C01854=-39.047,41.696,70.261,-152.7994,22.7901,0.0000
C01855=-37.223,43.443,70.297,-153.2837,23.1916,0.0000
C01856=-35.654,46.271,71.114,-156.3959,25.4216,0.0000
C01857=-37.003,49.553,73.167,-158.5816,26.4914,0.0000
C01858=-40.330,54.011,75.971,-161.3962,27.5073,0.0000
C01859=-44.783,59.707,78.794,-168.9608,27.8156,0.0000
C01860=-49.635,65.937,80.892,179.6697,0.5804,0.0000
C01861=-53.873,71.781,81.904,-177.7544,-3.3917,0.0000
C01862=-55.051,77.964,82.431,-176.8237,-4.6670,0.0000
C01863=-52.900,83.695,82.857,-176.4241,-5.2464,0.0000
C01864=-47.863,87.788,83.283,-176.3779,-5.3278,0.0000
C01865=-41.570,90.949,83.562,-176.4970,-5.1678,0.0000
C01866=-34.916,93.705,83.562,178.8092,6.1263,0.0000
C01867=-28.231,95.920,83.283,178.7790,6.3232,0.0000
C01868=-21.776,96.587,82.857,178.8046,6.2332,0.0000
C01869=-16.202,94.056,82.431,178.9359,5.5425,0.0000
